Fanuc TP program (LS listing): hs_ov_schraeg2.ls

/PROG  hs_ov_schraeg2
/ATTR
COMMENT	= "18-08-13 11:43:22";
PROG_SIZE	= 0;
DEFAULT_GROUP	= 1, 1, *, *, *;
/APPL
    ARC Welding Equipment: 1, *, *, *, *;
/MN
   1:  CALL HOME_ALL;
   1:  UFRAME_NUM = 1;
   1:  UTOOL_NUM = 3;
   1:  COL GUARD ADJUST 150;
   1:  PR[91] = PR[90];
   1:  ! Sicherheitspunkt;
   1:  PR[92] = PR[90];
   1:  PR[92] = PR[GP1:92,3] + 50;
   1:J PR[92];
   1:  PR[GP1:91,1] = PR[GP1:90,1] + 5.219;
   1:  PR[GP1:91,2] = PR[GP1:90,2] + -0.246;
   1:  PR[GP1:91,3] = PR[GP1:90,3] + 0.915;
   1:L PR[91] 10mm/sec CNT100;
   1:  PR[GP1:91,1] = PR[GP1:90,1] + 8.951;
   1:  PR[GP1:91,2] = PR[GP1:90,2] + -14.614;
   1:L PR[91] 10mm/sec CNT100;
   1:  PR[GP1:91,1] = PR[GP1:90,1] + 8.999;
   1:  PR[GP1:91,2] = PR[GP1:90,2] + -14.812;
   1:L PR[91] 10mm/sec CNT100;
   1:  PR[GP1:91,1] = PR[GP1:90,1] + 9.060;
   1:  PR[GP1:91,2] = PR[GP1:90,2] + -15.209;
   1:L PR[91] 10mm/sec CNT100;
   1:  PR[GP1:91,1] = PR[GP1:90,1] + 9.161;
   1:  PR[GP1:91,2] = PR[GP1:90,2] + -15.468;
   1:L PR[91] 10mm/sec CNT100;
   1:  PR[GP1:91,1] = PR[GP1:90,1] + 18.462;
   1:  PR[GP1:91,2] = PR[GP1:90,2] + -26.550;
   1:L PR[91] 10mm/sec CNT100;
   1:  PR[GP1:91,1] = PR[GP1:90,1] + 18.690;
   1:  PR[GP1:91,2] = PR[GP1:90,2] + -26.887;
   1:L PR[91] 10mm/sec CNT100;
   1:  PR[GP1:91,1] = PR[GP1:90,1] + 18.892;
   1:  PR[GP1:91,2] = PR[GP1:90,2] + -27.077;
   1:L PR[91] 10mm/sec CNT100;
   1:  PR[GP1:91,1] = PR[GP1:90,1] + 32.055;
   1:  PR[GP1:91,2] = PR[GP1:90,2] + -33.088;
   1:L PR[91] 10mm/sec CNT100;
   1:  PR[GP1:91,1] = PR[GP1:90,1] + 32.405;
   1:  PR[GP1:91,2] = PR[GP1:90,2] + -33.295;
   1:L PR[91] 10mm/sec CNT100;
   1:  PR[GP1:91,1] = PR[GP1:90,1] + 32.669;
   1:  PR[GP1:91,2] = PR[GP1:90,2] + -33.380;
   1:L PR[91] 10mm/sec CNT100;
   1:  PR[GP1:91,1] = PR[GP1:90,1] + 47.143;
   1:  PR[GP1:91,2] = PR[GP1:90,2] + -33.149;
   1:L PR[91] 10mm/sec CNT100;
   1:  PR[GP1:91,1] = PR[GP1:90,1] + 47.549;
   1:  PR[GP1:91,2] = PR[GP1:90,2] + -33.186;
   1:L PR[91] 10mm/sec CNT100;
   1:  PR[GP1:91,1] = PR[GP1:90,1] + 47.822;
   1:  PR[GP1:91,2] = PR[GP1:90,2] + -33.150;
   1:L PR[91] 10mm/sec CNT100;
   1:  PR[GP1:91,1] = PR[GP1:90,1] + 60.787;
   1:  PR[GP1:91,2] = PR[GP1:90,2] + -26.722;
   1:L PR[91] 10mm/sec CNT100;
   1:  PR[GP1:91,1] = PR[GP1:90,1] + 61.170;
   1:  PR[GP1:91,2] = PR[GP1:90,2] + -26.581;
   1:L PR[91] 10mm/sec CNT100;
   1:  PR[GP1:91,1] = PR[GP1:90,1] + 61.401;
   1:  PR[GP1:91,2] = PR[GP1:90,2] + -26.432;
   1:L PR[91] 10mm/sec CNT100;
   1:  PR[GP1:91,1] = PR[GP1:90,1] + 70.346;
   1:  PR[GP1:91,2] = PR[GP1:90,2] + -15.058;
   1:L PR[91] 10mm/sec CNT100;
   1:  PR[GP1:91,1] = PR[GP1:90,1] + 70.631;
   1:  PR[GP1:91,2] = PR[GP1:90,2] + -14.767;
   1:L PR[91] 10mm/sec CNT100;
   1:  PR[GP1:91,1] = PR[GP1:90,1] + 70.776;
   1:  PR[GP1:91,2] = PR[GP1:90,2] + -14.533;
   1:L PR[91] 10mm/sec CNT100;
   1:  PR[GP1:91,1] = PR[GP1:90,1] + 73.966;
   1:  PR[GP1:91,2] = PR[GP1:90,2] + -0.414;
   1:L PR[91] 10mm/sec CNT100;
   1:  PR[GP1:91,1] = PR[GP1:90,1] + 74.099;
   1:  PR[GP1:91,2] = PR[GP1:90,2] + -0.028;
   1:L PR[91] 10mm/sec CNT100;
   1:  PR[GP1:91,1] = PR[GP1:90,1] + 74.129;
   1:  PR[GP1:91,2] = PR[GP1:90,2] + 0.245;
   1:L PR[91] 10mm/sec CNT100;
   1:  PR[GP1:91,1] = PR[GP1:90,1] + 70.940;
   1:  PR[GP1:91,2] = PR[GP1:90,2] + 14.363;
   1:L PR[91] 10mm/sec CNT100;
   1:  PR[GP1:91,1] = PR[GP1:90,1] + 70.895;
   1:  PR[GP1:91,2] = PR[GP1:90,2] + 14.770;
   1:L PR[91] 10mm/sec CNT100;
   1:  PR[GP1:91,1] = PR[GP1:90,1] + 70.794;
   1:  PR[GP1:91,2] = PR[GP1:90,2] + 15.062;
   1:L PR[91] 10mm/sec CNT100;
   1:  PR[GP1:91,1] = PR[GP1:90,1] + 70.614;
   1:  PR[GP1:91,2] = PR[GP1:90,2] + 15.353;
   1:L PR[91] 10mm/sec CNT100;
   1:  PR[GP1:91,1] = PR[GP1:90,1] + 61.669;
   1:  PR[GP1:91,2] = PR[GP1:90,2] + 26.727;
   1:L PR[91] 10mm/sec CNT100;
   1:  PR[GP1:91,1] = PR[GP1:90,1] + 61.429;
   1:  PR[GP1:91,2] = PR[GP1:90,2] + 26.972;
   1:L PR[91] 10mm/sec CNT100;
   1:  PR[GP1:91,1] = PR[GP1:90,1] + 61.143;
   1:  PR[GP1:91,2] = PR[GP1:90,2] + 27.157;
   1:L PR[91] 10mm/sec CNT100;
   1:  PR[GP1:91,1] = PR[GP1:90,1] + 48.177;
   1:  PR[GP1:91,2] = PR[GP1:90,2] + 33.585;
   1:L PR[91] 10mm/sec CNT100;
   1:  PR[GP1:91,1] = PR[GP1:90,1] + 47.855;
   1:  PR[GP1:91,2] = PR[GP1:90,2] + 33.703;
   1:L PR[91] 10mm/sec CNT100;
   1:  PR[GP1:91,1] = PR[GP1:90,1] + 47.517;
   1:  PR[GP1:91,2] = PR[GP1:90,2] + 33.748;
   1:L PR[91] 10mm/sec CNT100;
   1:  PR[GP1:91,1] = PR[GP1:90,1] + 33.042;
   1:  PR[GP1:91,2] = PR[GP1:90,2] + 33.978;
   1:L PR[91] 10mm/sec CNT100;
   1:  PR[GP1:91,1] = PR[GP1:90,1] + 32.700;
   1:  PR[GP1:91,2] = PR[GP1:90,2] + 33.948;
   1:L PR[91] 10mm/sec CNT100;
   1:  PR[GP1:91,1] = PR[GP1:90,1] + 32.375;
   1:  PR[GP1:91,2] = PR[GP1:90,2] + 33.843;
   1:L PR[91] 10mm/sec CNT100;
   1:  PR[GP1:91,1] = PR[GP1:90,1] + 19.212;
   1:  PR[GP1:91,2] = PR[GP1:90,2] + 27.832;
   1:L PR[91] 10mm/sec CNT100;
   1:  PR[GP1:91,1] = PR[GP1:90,1] + 18.915;
   1:  PR[GP1:91,2] = PR[GP1:90,2] + 27.657;
   1:L PR[91] 10mm/sec CNT100;
   1:  PR[GP1:91,1] = PR[GP1:90,1] + 18.668;
   1:  PR[GP1:91,2] = PR[GP1:90,2] + 27.424;
   1:L PR[91] 10mm/sec CNT100;
   1:  PR[GP1:91,1] = PR[GP1:90,1] + 9.365;
   1:  PR[GP1:91,2] = PR[GP1:90,2] + 16.341;
   1:L PR[91] 10mm/sec CNT100;
   1:  PR[GP1:91,1] = PR[GP1:90,1] + 9.172;
   1:  PR[GP1:91,2] = PR[GP1:90,2] + 16.055;
   1:L PR[91] 10mm/sec CNT100;
   1:  PR[GP1:91,1] = PR[GP1:90,1] + 9.048;
   1:  PR[GP1:91,2] = PR[GP1:90,2] + 15.739;
   1:L PR[91] 10mm/sec CNT100;
   1:  PR[GP1:91,1] = PR[GP1:90,1] + 5.411;
   1:  PR[GP1:91,2] = PR[GP1:90,2] + 1.740;
   1:L PR[91] 10mm/sec CNT100;
   1:  PR[GP1:91,1] = PR[GP1:90,1] + 5.272;
   1:  PR[GP1:91,2] = PR[GP1:90,2] + 0.804;
   1:L PR[91] 10mm/sec CNT100;
   1:  PR[GP1:91,1] = PR[GP1:90,1] + -5.745;
   1:L PR[91] 10mm/sec CNT100;
   1:  PR[GP1:91,1] = PR[GP1:90,1] + -9.477;
   1:  PR[GP1:91,2] = PR[GP1:90,2] + 15.172;
   1:L PR[91] 10mm/sec CNT100;
   1:  PR[GP1:91,1] = PR[GP1:90,1] + -9.525;
   1:  PR[GP1:91,2] = PR[GP1:90,2] + 15.371;
   1:L PR[91] 10mm/sec CNT100;
   1:  PR[GP1:91,1] = PR[GP1:90,1] + -9.586;
   1:  PR[GP1:91,2] = PR[GP1:90,2] + 15.768;
   1:L PR[91] 10mm/sec CNT100;
   1:  PR[GP1:91,1] = PR[GP1:90,1] + -9.687;
   1:  PR[GP1:91,2] = PR[GP1:90,2] + 16.026;
   1:L PR[91] 10mm/sec CNT100;
   1:  PR[GP1:91,1] = PR[GP1:90,1] + -18.989;
   1:  PR[GP1:91,2] = PR[GP1:90,2] + 27.108;
   1:L PR[91] 10mm/sec CNT100;
   1:  PR[GP1:91,1] = PR[GP1:90,1] + -19.217;
   1:  PR[GP1:91,2] = PR[GP1:90,2] + 27.445;
   1:L PR[91] 10mm/sec CNT100;
   1:  PR[GP1:91,1] = PR[GP1:90,1] + -19.418;
   1:  PR[GP1:91,2] = PR[GP1:90,2] + 27.635;
   1:L PR[91] 10mm/sec CNT100;
   1:  PR[GP1:91,1] = PR[GP1:90,1] + -32.581;
   1:  PR[GP1:91,2] = PR[GP1:90,2] + 33.646;
   1:L PR[91] 10mm/sec CNT100;
   1:  PR[GP1:91,1] = PR[GP1:90,1] + -32.932;
   1:  PR[GP1:91,2] = PR[GP1:90,2] + 33.853;
   1:L PR[91] 10mm/sec CNT100;
   1:  PR[GP1:91,1] = PR[GP1:90,1] + -33.195;
   1:  PR[GP1:91,2] = PR[GP1:90,2] + 33.938;
   1:L PR[91] 10mm/sec CNT100;
   1:  PR[GP1:91,1] = PR[GP1:90,1] + -47.669;
   1:  PR[GP1:91,2] = PR[GP1:90,2] + 33.707;
   1:L PR[91] 10mm/sec CNT100;
   1:  PR[GP1:91,1] = PR[GP1:90,1] + -48.075;
   1:  PR[GP1:91,2] = PR[GP1:90,2] + 33.744;
   1:L PR[91] 10mm/sec CNT100;
   1:  PR[GP1:91,1] = PR[GP1:90,1] + -48.349;
   1:  PR[GP1:91,2] = PR[GP1:90,2] + 33.708;
   1:L PR[91] 10mm/sec CNT100;
   1:  PR[GP1:91,1] = PR[GP1:90,1] + -61.314;
   1:  PR[GP1:91,2] = PR[GP1:90,2] + 27.280;
   1:L PR[91] 10mm/sec CNT100;
   1:  PR[GP1:91,1] = PR[GP1:90,1] + -61.696;
   1:  PR[GP1:91,2] = PR[GP1:90,2] + 27.140;
   1:L PR[91] 10mm/sec CNT100;
   1:  PR[GP1:91,1] = PR[GP1:90,1] + -61.928;
   1:  PR[GP1:91,2] = PR[GP1:90,2] + 26.990;
   1:L PR[91] 10mm/sec CNT100;
   1:  PR[GP1:91,1] = PR[GP1:90,1] + -70.872;
   1:  PR[GP1:91,2] = PR[GP1:90,2] + 15.617;
   1:L PR[91] 10mm/sec CNT100;
   1:  PR[GP1:91,1] = PR[GP1:90,1] + -71.158;
   1:  PR[GP1:91,2] = PR[GP1:90,2] + 15.325;
   1:L PR[91] 10mm/sec CNT100;
   1:  PR[GP1:91,1] = PR[GP1:90,1] + -71.303;
   1:  PR[GP1:91,2] = PR[GP1:90,2] + 15.091;
   1:L PR[91] 10mm/sec CNT100;
   1:  PR[GP1:91,1] = PR[GP1:90,1] + -74.492;
   1:  PR[GP1:91,2] = PR[GP1:90,2] + 0.972;
   1:L PR[91] 10mm/sec CNT100;
   1:  PR[GP1:91,1] = PR[GP1:90,1] + -74.625;
   1:  PR[GP1:91,2] = PR[GP1:90,2] + 0.586;
   1:L PR[91] 10mm/sec CNT100;
   1:  PR[GP1:91,1] = PR[GP1:90,1] + -74.656;
   1:  PR[GP1:91,2] = PR[GP1:90,2] + 0.313;
   1:L PR[91] 10mm/sec CNT100;
   1:  PR[GP1:91,1] = PR[GP1:90,1] + -71.466;
   1:  PR[GP1:91,2] = PR[GP1:90,2] + -13.805;
   1:L PR[91] 10mm/sec CNT100;
   1:  PR[GP1:91,1] = PR[GP1:90,1] + -71.421;
   1:  PR[GP1:91,2] = PR[GP1:90,2] + -14.212;
   1:L PR[91] 10mm/sec CNT100;
   1:  PR[GP1:91,1] = PR[GP1:90,1] + -71.320;
   1:  PR[GP1:91,2] = PR[GP1:90,2] + -14.504;
   1:L PR[91] 10mm/sec CNT100;
   1:  PR[GP1:91,1] = PR[GP1:90,1] + -71.141;
   1:  PR[GP1:91,2] = PR[GP1:90,2] + -14.795;
   1:L PR[91] 10mm/sec CNT100;
   1:  PR[GP1:91,1] = PR[GP1:90,1] + -62.196;
   1:  PR[GP1:91,2] = PR[GP1:90,2] + -26.169;
   1:L PR[91] 10mm/sec CNT100;
   1:  PR[GP1:91,1] = PR[GP1:90,1] + -61.956;
   1:  PR[GP1:91,2] = PR[GP1:90,2] + -26.414;
   1:L PR[91] 10mm/sec CNT100;
   1:  PR[GP1:91,1] = PR[GP1:90,1] + -61.669;
   1:  PR[GP1:91,2] = PR[GP1:90,2] + -26.599;
   1:L PR[91] 10mm/sec CNT100;
   1:  PR[GP1:91,1] = PR[GP1:90,1] + -48.703;
   1:  PR[GP1:91,2] = PR[GP1:90,2] + -33.027;
   1:L PR[91] 10mm/sec CNT100;
   1:  PR[GP1:91,1] = PR[GP1:90,1] + -48.381;
   1:  PR[GP1:91,2] = PR[GP1:90,2] + -33.145;
   1:L PR[91] 10mm/sec CNT100;
   1:  PR[GP1:91,1] = PR[GP1:90,1] + -48.043;
   1:  PR[GP1:91,2] = PR[GP1:90,2] + -33.190;
   1:L PR[91] 10mm/sec CNT100;
   1:  PR[GP1:91,1] = PR[GP1:90,1] + -33.568;
   1:  PR[GP1:91,2] = PR[GP1:90,2] + -33.420;
   1:L PR[91] 10mm/sec CNT100;
   1:  PR[GP1:91,1] = PR[GP1:90,1] + -33.226;
   1:  PR[GP1:91,2] = PR[GP1:90,2] + -33.390;
   1:L PR[91] 10mm/sec CNT100;
   1:  PR[GP1:91,1] = PR[GP1:90,1] + -32.902;
   1:  PR[GP1:91,2] = PR[GP1:90,2] + -33.285;
   1:L PR[91] 10mm/sec CNT100;
   1:  PR[GP1:91,1] = PR[GP1:90,1] + -19.738;
   1:  PR[GP1:91,2] = PR[GP1:90,2] + -27.274;
   1:L PR[91] 10mm/sec CNT100;
   1:  PR[GP1:91,1] = PR[GP1:90,1] + -19.442;
   1:  PR[GP1:91,2] = PR[GP1:90,2] + -27.099;
   1:L PR[91] 10mm/sec CNT100;
   1:  PR[GP1:91,1] = PR[GP1:90,1] + -19.194;
   1:  PR[GP1:91,2] = PR[GP1:90,2] + -26.866;
   1:L PR[91] 10mm/sec CNT100;
   1:  PR[GP1:91,1] = PR[GP1:90,1] + -9.892;
   1:  PR[GP1:91,2] = PR[GP1:90,2] + -15.783;
   1:L PR[91] 10mm/sec CNT100;
   1:  PR[GP1:91,1] = PR[GP1:90,1] + -9.699;
   1:  PR[GP1:91,2] = PR[GP1:90,2] + -15.497;
   1:L PR[91] 10mm/sec CNT100;
   1:  PR[GP1:91,1] = PR[GP1:90,1] + -9.575;
   1:  PR[GP1:91,2] = PR[GP1:90,2] + -15.181;
   1:L PR[91] 10mm/sec CNT100;
   1:  PR[GP1:91,1] = PR[GP1:90,1] + -5.938;
   1:  PR[GP1:91,2] = PR[GP1:90,2] + -1.182;
   1:L PR[91] 10mm/sec CNT100;
   1:  PR[GP1:91,1] = PR[GP1:90,1] + -5.799;
   1:  PR[GP1:91,2] = PR[GP1:90,2] + -0.246;
   1:L PR[91] 10mm/sec CNT100;
   1:  PR[GP1:91,1] = PR[GP1:90,1] + 5.219;
   1:L PR[91] 10mm/sec CNT100;
   1:  PR[GP1:91,1] = PR[GP1:90,1] + 8.514;
   1:  PR[GP1:91,2] = PR[GP1:90,2] + -12.941;
   1:  PR[GP1:91,3] = PR[GP1:90,3] + 1.525;
   1:L PR[91] 10mm/sec CNT100;
   1:  PR[GP1:91,1] = PR[GP1:90,1] + 8.631;
   1:  PR[GP1:91,2] = PR[GP1:90,2] + -13.421;
   1:L PR[91] 10mm/sec CNT100;
   1:  PR[GP1:91,1] = PR[GP1:90,1] + 8.803;
   1:  PR[GP1:91,2] = PR[GP1:90,2] + -14.547;
   1:L PR[91] 10mm/sec CNT100;
   1:  PR[GP1:91,1] = PR[GP1:90,1] + 9.173;
   1:  PR[GP1:91,2] = PR[GP1:90,2] + -15.491;
   1:L PR[91] 10mm/sec CNT100;
   1:  PR[GP1:91,1] = PR[GP1:90,1] + 17.530;
   1:  PR[GP1:91,2] = PR[GP1:90,2] + -25.448;
   1:L PR[91] 10mm/sec CNT100;
   1:  PR[GP1:91,1] = PR[GP1:90,1] + 18.171;
   1:  PR[GP1:91,2] = PR[GP1:90,2] + -26.396;
   1:L PR[91] 10mm/sec CNT100;
   1:  PR[GP1:91,1] = PR[GP1:90,1] + 18.910;
   1:  PR[GP1:91,2] = PR[GP1:90,2] + -27.090;
   1:L PR[91] 10mm/sec CNT100;
   1:  PR[GP1:91,1] = PR[GP1:90,1] + 30.736;
   1:  PR[GP1:91,2] = PR[GP1:90,2] + -32.491;
   1:L PR[91] 10mm/sec CNT100;
   1:  PR[GP1:91,1] = PR[GP1:90,1] + 31.721;
   1:  PR[GP1:91,2] = PR[GP1:90,2] + -33.072;
   1:L PR[91] 10mm/sec CNT100;
   1:  PR[GP1:91,1] = PR[GP1:90,1] + 32.686;
   1:  PR[GP1:91,2] = PR[GP1:90,2] + -33.383;
   1:L PR[91] 10mm/sec CNT100;
   1:  PR[GP1:91,1] = PR[GP1:90,1] + 45.690;
   1:  PR[GP1:91,2] = PR[GP1:90,2] + -33.176;
   1:L PR[91] 10mm/sec CNT100;
   1:  PR[GP1:91,1] = PR[GP1:90,1] + 46.831;
   1:  PR[GP1:91,2] = PR[GP1:90,2] + -33.279;
   1:L PR[91] 10mm/sec CNT100;
   1:  PR[GP1:91,1] = PR[GP1:90,1] + 47.835;
   1:  PR[GP1:91,2] = PR[GP1:90,2] + -33.147;
   1:L PR[91] 10mm/sec CNT100;
   1:  PR[GP1:91,1] = PR[GP1:90,1] + 59.483;
   1:  PR[GP1:91,2] = PR[GP1:90,2] + -27.372;
   1:L PR[91] 10mm/sec CNT100;
   1:  PR[GP1:91,1] = PR[GP1:90,1] + 60.558;
   1:  PR[GP1:91,2] = PR[GP1:90,2] + -26.976;
   1:L PR[91] 10mm/sec CNT100;
   1:  PR[GP1:91,1] = PR[GP1:90,1] + 61.408;
   1:  PR[GP1:91,2] = PR[GP1:90,2] + -26.426;
   1:L PR[91] 10mm/sec CNT100;
   1:  PR[GP1:91,1] = PR[GP1:90,1] + 69.444;
   1:  PR[GP1:91,2] = PR[GP1:90,2] + -16.208;
   1:L PR[91] 10mm/sec CNT100;
   1:  PR[GP1:91,1] = PR[GP1:90,1] + 70.246;
   1:  PR[GP1:91,2] = PR[GP1:90,2] + -15.390;
   1:L PR[91] 10mm/sec CNT100;
   1:  PR[GP1:91,1] = PR[GP1:90,1] + 70.778;
   1:  PR[GP1:91,2] = PR[GP1:90,2] + -14.528;
   1:L PR[91] 10mm/sec CNT100;
   1:  PR[GP1:91,1] = PR[GP1:90,1] + 73.644;
   1:  PR[GP1:91,2] = PR[GP1:90,2] + -1.844;
   1:L PR[91] 10mm/sec CNT100;
   1:  PR[GP1:91,1] = PR[GP1:90,1] + 74.018;
   1:  PR[GP1:91,2] = PR[GP1:90,2] + -0.761;
   1:L PR[91] 10mm/sec CNT100;
   1:  PR[GP1:91,1] = PR[GP1:90,1] + 74.129;
   1:  PR[GP1:91,2] = PR[GP1:90,2] + 0.245;
   1:L PR[91] 10mm/sec CNT100;
   1:  PR[GP1:91,1] = PR[GP1:90,1] + 71.264;
   1:  PR[GP1:91,2] = PR[GP1:90,2] + 12.930;
   1:L PR[91] 10mm/sec CNT100;
   1:  PR[GP1:91,1] = PR[GP1:90,1] + 71.137;
   1:  PR[GP1:91,2] = PR[GP1:90,2] + 14.069;
   1:L PR[91] 10mm/sec CNT100;
   1:  PR[GP1:91,1] = PR[GP1:90,1] + 70.796;
   1:  PR[GP1:91,2] = PR[GP1:90,2] + 15.058;
   1:L PR[91] 10mm/sec CNT100;
   1:  PR[GP1:91,1] = PR[GP1:90,1] + 70.229;
   1:  PR[GP1:91,2] = PR[GP1:90,2] + 15.976;
   1:L PR[91] 10mm/sec CNT100;
   1:  PR[GP1:91,1] = PR[GP1:90,1] + 62.192;
   1:  PR[GP1:91,2] = PR[GP1:90,2] + 26.195;
   1:L PR[91] 10mm/sec CNT100;
   1:  PR[GP1:91,1] = PR[GP1:90,1] + 61.436;
   1:  PR[GP1:91,2] = PR[GP1:90,2] + 26.966;
   1:L PR[91] 10mm/sec CNT100;
   1:  PR[GP1:91,1] = PR[GP1:90,1] + 60.531;
   1:  PR[GP1:91,2] = PR[GP1:90,2] + 27.552;
   1:L PR[91] 10mm/sec CNT100;
   1:  PR[GP1:91,1] = PR[GP1:90,1] + 48.882;
   1:  PR[GP1:91,2] = PR[GP1:90,2] + 33.327;
   1:L PR[91] 10mm/sec CNT100;
   1:  PR[GP1:91,1] = PR[GP1:90,1] + 47.868;
   1:  PR[GP1:91,2] = PR[GP1:90,2] + 33.700;
   1:L PR[91] 10mm/sec CNT100;
   1:  PR[GP1:91,1] = PR[GP1:90,1] + 46.799;
   1:  PR[GP1:91,2] = PR[GP1:90,2] + 33.842;
   1:L PR[91] 10mm/sec CNT100;
   1:  PR[GP1:91,1] = PR[GP1:90,1] + 33.794;
   1:  PR[GP1:91,2] = PR[GP1:90,2] + 34.049;
   1:L PR[91] 10mm/sec CNT100;
   1:  PR[GP1:91,1] = PR[GP1:90,1] + 32.717;
   1:  PR[GP1:91,2] = PR[GP1:90,2] + 33.951;
   1:L PR[91] 10mm/sec CNT100;
   1:  PR[GP1:91,1] = PR[GP1:90,1] + 31.691;
   1:  PR[GP1:91,2] = PR[GP1:90,2] + 33.621;
   1:L PR[91] 10mm/sec CNT100;
   1:  PR[GP1:91,1] = PR[GP1:90,1] + 19.865;
   1:  PR[GP1:91,2] = PR[GP1:90,2] + 28.220;
   1:L PR[91] 10mm/sec CNT100;
   1:  PR[GP1:91,1] = PR[GP1:90,1] + 18.933;
   1:  PR[GP1:91,2] = PR[GP1:90,2] + 27.670;
   1:L PR[91] 10mm/sec CNT100;
   1:  PR[GP1:91,1] = PR[GP1:90,1] + 18.148;
   1:  PR[GP1:91,2] = PR[GP1:90,2] + 26.932;
   1:L PR[91] 10mm/sec CNT100;
   1:  PR[GP1:91,1] = PR[GP1:90,1] + 9.791;
   1:  PR[GP1:91,2] = PR[GP1:90,2] + 16.975;
   1:L PR[91] 10mm/sec CNT100;
   1:  PR[GP1:91,1] = PR[GP1:90,1] + 9.185;
   1:  PR[GP1:91,2] = PR[GP1:90,2] + 16.079;
   1:L PR[91] 10mm/sec CNT100;
   1:  PR[GP1:91,1] = PR[GP1:90,1] + 8.792;
   1:  PR[GP1:91,2] = PR[GP1:90,2] + 15.076;
   1:L PR[91] 10mm/sec CNT100;
   1:  PR[GP1:91,1] = PR[GP1:90,1] + 5.524;
   1:  PR[GP1:91,2] = PR[GP1:90,2] + 2.499;
   1:L PR[91] 10mm/sec CNT100;
   1:  PR[GP1:91,1] = PR[GP1:90,1] + 5.272;
   1:  PR[GP1:91,2] = PR[GP1:90,2] + 0.804;
   1:L PR[91] 10mm/sec CNT100;
   1:  PR[GP1:91,1] = PR[GP1:90,1] + -5.745;
   1:L PR[91] 10mm/sec CNT100;
   1:  PR[GP1:91,1] = PR[GP1:90,1] + -9.040;
   1:  PR[GP1:91,2] = PR[GP1:90,2] + 13.499;
   1:L PR[91] 10mm/sec CNT100;
   1:  PR[GP1:91,1] = PR[GP1:90,1] + -9.157;
   1:  PR[GP1:91,2] = PR[GP1:90,2] + 13.979;
   1:L PR[91] 10mm/sec CNT100;
   1:  PR[GP1:91,1] = PR[GP1:90,1] + -9.329;
   1:  PR[GP1:91,2] = PR[GP1:90,2] + 15.105;
   1:L PR[91] 10mm/sec CNT100;
   1:  PR[GP1:91,1] = PR[GP1:90,1] + -9.699;
   1:  PR[GP1:91,2] = PR[GP1:90,2] + 16.049;
   1:L PR[91] 10mm/sec CNT100;
   1:  PR[GP1:91,1] = PR[GP1:90,1] + -18.056;
   1:  PR[GP1:91,2] = PR[GP1:90,2] + 26.006;
   1:L PR[91] 10mm/sec CNT100;
   1:  PR[GP1:91,1] = PR[GP1:90,1] + -18.697;
   1:  PR[GP1:91,2] = PR[GP1:90,2] + 26.954;
   1:L PR[91] 10mm/sec CNT100;
   1:  PR[GP1:91,1] = PR[GP1:90,1] + -19.436;
   1:  PR[GP1:91,2] = PR[GP1:90,2] + 27.648;
   1:L PR[91] 10mm/sec CNT100;
   1:  PR[GP1:91,1] = PR[GP1:90,1] + -31.262;
   1:  PR[GP1:91,2] = PR[GP1:90,2] + 33.049;
   1:L PR[91] 10mm/sec CNT100;
   1:  PR[GP1:91,1] = PR[GP1:90,1] + -32.248;
   1:  PR[GP1:91,2] = PR[GP1:90,2] + 33.631;
   1:L PR[91] 10mm/sec CNT100;
   1:  PR[GP1:91,1] = PR[GP1:90,1] + -33.213;
   1:  PR[GP1:91,2] = PR[GP1:90,2] + 33.941;
   1:L PR[91] 10mm/sec CNT100;
   1:  PR[GP1:91,1] = PR[GP1:90,1] + -46.217;
   1:  PR[GP1:91,2] = PR[GP1:90,2] + 33.734;
   1:L PR[91] 10mm/sec CNT100;
   1:  PR[GP1:91,1] = PR[GP1:90,1] + -47.357;
   1:  PR[GP1:91,2] = PR[GP1:90,2] + 33.837;
   1:L PR[91] 10mm/sec CNT100;
   1:  PR[GP1:91,1] = PR[GP1:90,1] + -48.361;
   1:  PR[GP1:91,2] = PR[GP1:90,2] + 33.705;
   1:L PR[91] 10mm/sec CNT100;
   1:  PR[GP1:91,1] = PR[GP1:90,1] + -60.010;
   1:  PR[GP1:91,2] = PR[GP1:90,2] + 27.930;
   1:L PR[91] 10mm/sec CNT100;
   1:  PR[GP1:91,1] = PR[GP1:90,1] + -61.084;
   1:  PR[GP1:91,2] = PR[GP1:90,2] + 27.534;
   1:L PR[91] 10mm/sec CNT100;
   1:  PR[GP1:91,1] = PR[GP1:90,1] + -61.935;
   1:  PR[GP1:91,2] = PR[GP1:90,2] + 26.984;
   1:L PR[91] 10mm/sec CNT100;
   1:  PR[GP1:91,1] = PR[GP1:90,1] + -69.971;
   1:  PR[GP1:91,2] = PR[GP1:90,2] + 16.766;
   1:L PR[91] 10mm/sec CNT100;
   1:  PR[GP1:91,1] = PR[GP1:90,1] + -70.772;
   1:  PR[GP1:91,2] = PR[GP1:90,2] + 15.948;
   1:L PR[91] 10mm/sec CNT100;
   1:  PR[GP1:91,1] = PR[GP1:90,1] + -71.305;
   1:  PR[GP1:91,2] = PR[GP1:90,2] + 15.087;
   1:L PR[91] 10mm/sec CNT100;
   1:  PR[GP1:91,1] = PR[GP1:90,1] + -74.170;
   1:  PR[GP1:91,2] = PR[GP1:90,2] + 2.402;
   1:L PR[91] 10mm/sec CNT100;
   1:  PR[GP1:91,1] = PR[GP1:90,1] + -74.544;
   1:  PR[GP1:91,2] = PR[GP1:90,2] + 1.319;
   1:L PR[91] 10mm/sec CNT100;
   1:  PR[GP1:91,1] = PR[GP1:90,1] + -74.656;
   1:  PR[GP1:91,2] = PR[GP1:90,2] + 0.313;
   1:L PR[91] 10mm/sec CNT100;
   1:  PR[GP1:91,1] = PR[GP1:90,1] + -71.790;
   1:  PR[GP1:91,2] = PR[GP1:90,2] + -12.371;
   1:L PR[91] 10mm/sec CNT100;
   1:  PR[GP1:91,1] = PR[GP1:90,1] + -71.663;
   1:  PR[GP1:91,2] = PR[GP1:90,2] + -13.511;
   1:L PR[91] 10mm/sec CNT100;
   1:  PR[GP1:91,1] = PR[GP1:90,1] + -71.322;
   1:  PR[GP1:91,2] = PR[GP1:90,2] + -14.500;
   1:L PR[91] 10mm/sec CNT100;
   1:  PR[GP1:91,1] = PR[GP1:90,1] + -70.755;
   1:  PR[GP1:91,2] = PR[GP1:90,2] + -15.418;
   1:L PR[91] 10mm/sec CNT100;
   1:  PR[GP1:91,1] = PR[GP1:90,1] + -62.719;
   1:  PR[GP1:91,2] = PR[GP1:90,2] + -25.636;
   1:L PR[91] 10mm/sec CNT100;
   1:  PR[GP1:91,1] = PR[GP1:90,1] + -61.963;
   1:  PR[GP1:91,2] = PR[GP1:90,2] + -26.408;
   1:L PR[91] 10mm/sec CNT100;
   1:  PR[GP1:91,1] = PR[GP1:90,1] + -61.057;
   1:  PR[GP1:91,2] = PR[GP1:90,2] + -26.994;
   1:L PR[91] 10mm/sec CNT100;
   1:  PR[GP1:91,1] = PR[GP1:90,1] + -49.408;
   1:  PR[GP1:91,2] = PR[GP1:90,2] + -32.769;
   1:L PR[91] 10mm/sec CNT100;
   1:  PR[GP1:91,1] = PR[GP1:90,1] + -48.394;
   1:  PR[GP1:91,2] = PR[GP1:90,2] + -33.142;
   1:L PR[91] 10mm/sec CNT100;
   1:  PR[GP1:91,1] = PR[GP1:90,1] + -47.325;
   1:  PR[GP1:91,2] = PR[GP1:90,2] + -33.283;
   1:L PR[91] 10mm/sec CNT100;
   1:  PR[GP1:91,1] = PR[GP1:90,1] + -34.320;
   1:  PR[GP1:91,2] = PR[GP1:90,2] + -33.490;
   1:L PR[91] 10mm/sec CNT100;
   1:  PR[GP1:91,1] = PR[GP1:90,1] + -33.244;
   1:  PR[GP1:91,2] = PR[GP1:90,2] + -33.393;
   1:L PR[91] 10mm/sec CNT100;
   1:  PR[GP1:91,1] = PR[GP1:90,1] + -32.218;
   1:  PR[GP1:91,2] = PR[GP1:90,2] + -33.063;
   1:L PR[91] 10mm/sec CNT100;
   1:  PR[GP1:91,1] = PR[GP1:90,1] + -20.391;
   1:  PR[GP1:91,2] = PR[GP1:90,2] + -27.662;
   1:L PR[91] 10mm/sec CNT100;
   1:  PR[GP1:91,1] = PR[GP1:90,1] + -19.460;
   1:  PR[GP1:91,2] = PR[GP1:90,2] + -27.112;
   1:L PR[91] 10mm/sec CNT100;
   1:  PR[GP1:91,1] = PR[GP1:90,1] + -18.675;
   1:  PR[GP1:91,2] = PR[GP1:90,2] + -26.374;
   1:L PR[91] 10mm/sec CNT100;
   1:  PR[GP1:91,1] = PR[GP1:90,1] + -10.317;
   1:  PR[GP1:91,2] = PR[GP1:90,2] + -16.417;
   1:L PR[91] 10mm/sec CNT100;
   1:  PR[GP1:91,1] = PR[GP1:90,1] + -9.711;
   1:  PR[GP1:91,2] = PR[GP1:90,2] + -15.521;
   1:L PR[91] 10mm/sec CNT100;
   1:  PR[GP1:91,1] = PR[GP1:90,1] + -9.318;
   1:  PR[GP1:91,2] = PR[GP1:90,2] + -14.518;
   1:L PR[91] 10mm/sec CNT100;
   1:  PR[GP1:91,1] = PR[GP1:90,1] + -6.050;
   1:  PR[GP1:91,2] = PR[GP1:90,2] + -1.940;
   1:L PR[91] 10mm/sec CNT100;
   1:  PR[GP1:91,1] = PR[GP1:90,1] + -5.799;
   1:  PR[GP1:91,2] = PR[GP1:90,2] + -0.246;
   1:L PR[91] 10mm/sec CNT100;
   1:  PR[GP1:91,1] = PR[GP1:90,1] + 5.219;
   1:L PR[91] 10mm/sec CNT100;
   1:  PR[GP1:91,1] = PR[GP1:90,1] + 8.164;
   1:  PR[GP1:91,2] = PR[GP1:90,2] + -11.602;
   1:  PR[GP1:91,3] = PR[GP1:90,3] + 2.135;
   1:L PR[91] 10mm/sec CNT100;
   1:  PR[GP1:91,1] = PR[GP1:90,1] + 8.336;
   1:  PR[GP1:91,2] = PR[GP1:90,2] + -12.307;
   1:L PR[91] 10mm/sec CNT100;
   1:  PR[GP1:91,1] = PR[GP1:90,1] + 8.598;
   1:  PR[GP1:91,2] = PR[GP1:90,2] + -14.016;
   1:L PR[91] 10mm/sec CNT100;
   1:  PR[GP1:91,1] = PR[GP1:90,1] + 9.183;
   1:  PR[GP1:91,2] = PR[GP1:90,2] + -15.510;
   1:L PR[91] 10mm/sec CNT100;
   1:  PR[GP1:91,1] = PR[GP1:90,1] + 16.784;
   1:  PR[GP1:91,2] = PR[GP1:90,2] + -24.567;
   1:L PR[91] 10mm/sec CNT100;
   1:  PR[GP1:91,1] = PR[GP1:90,1] + 17.756;
   1:  PR[GP1:91,2] = PR[GP1:90,2] + -26.002;
   1:L PR[91] 10mm/sec CNT100;
   1:  PR[GP1:91,1] = PR[GP1:90,1] + 18.924;
   1:  PR[GP1:91,2] = PR[GP1:90,2] + -27.101;
   1:L PR[91] 10mm/sec CNT100;
   1:  PR[GP1:91,1] = PR[GP1:90,1] + 29.681;
   1:  PR[GP1:91,2] = PR[GP1:90,2] + -32.013;
   1:L PR[91] 10mm/sec CNT100;
   1:  PR[GP1:91,1] = PR[GP1:90,1] + 31.174;
   1:  PR[GP1:91,2] = PR[GP1:90,2] + -32.895;
   1:L PR[91] 10mm/sec CNT100;
   1:  PR[GP1:91,1] = PR[GP1:90,1] + 32.701;
   1:  PR[GP1:91,2] = PR[GP1:90,2] + -33.386;
   1:L PR[91] 10mm/sec CNT100;
   1:  PR[GP1:91,1] = PR[GP1:90,1] + 44.529;
   1:  PR[GP1:91,2] = PR[GP1:90,2] + -33.198;
   1:L PR[91] 10mm/sec CNT100;
   1:  PR[GP1:91,1] = PR[GP1:90,1] + 46.256;
   1:  PR[GP1:91,2] = PR[GP1:90,2] + -33.354;
   1:L PR[91] 10mm/sec CNT100;
   1:  PR[GP1:91,1] = PR[GP1:90,1] + 47.845;
   1:  PR[GP1:91,2] = PR[GP1:90,2] + -33.144;
   1:L PR[91] 10mm/sec CNT100;
   1:  PR[GP1:91,1] = PR[GP1:90,1] + 58.440;
   1:  PR[GP1:91,2] = PR[GP1:90,2] + -27.892;
   1:L PR[91] 10mm/sec CNT100;
   1:  PR[GP1:91,1] = PR[GP1:90,1] + 60.068;
   1:  PR[GP1:91,2] = PR[GP1:90,2] + -27.292;
   1:L PR[91] 10mm/sec CNT100;
   1:  PR[GP1:91,1] = PR[GP1:90,1] + 61.414;
   1:  PR[GP1:91,2] = PR[GP1:90,2] + -26.422;
   1:L PR[91] 10mm/sec CNT100;
   1:  PR[GP1:91,1] = PR[GP1:90,1] + 68.723;
   1:  PR[GP1:91,2] = PR[GP1:90,2] + -17.128;
   1:L PR[91] 10mm/sec CNT100;
   1:  PR[GP1:91,1] = PR[GP1:90,1] + 69.937;
   1:  PR[GP1:91,2] = PR[GP1:90,2] + -15.888;
   1:L PR[91] 10mm/sec CNT100;
   1:  PR[GP1:91,1] = PR[GP1:90,1] + 70.780;
   1:  PR[GP1:91,2] = PR[GP1:90,2] + -14.525;
   1:L PR[91] 10mm/sec CNT100;
   1:  PR[GP1:91,1] = PR[GP1:90,1] + 73.386;
   1:  PR[GP1:91,2] = PR[GP1:90,2] + -2.988;
   1:L PR[91] 10mm/sec CNT100;
   1:  PR[GP1:91,1] = PR[GP1:90,1] + 73.952;
   1:  PR[GP1:91,2] = PR[GP1:90,2] + -1.347;
   1:L PR[91] 10mm/sec CNT100;
   1:  PR[GP1:91,1] = PR[GP1:90,1] + 74.129;
   1:  PR[GP1:91,2] = PR[GP1:90,2] + 0.245;
   1:L PR[91] 10mm/sec CNT100;
   1:  PR[GP1:91,1] = PR[GP1:90,1] + 71.523;
   1:  PR[GP1:91,2] = PR[GP1:90,2] + 11.782;
   1:L PR[91] 10mm/sec CNT100;
   1:  PR[GP1:91,1] = PR[GP1:90,1] + 71.331;
   1:  PR[GP1:91,2] = PR[GP1:90,2] + 13.508;
   1:L PR[91] 10mm/sec CNT100;
   1:  PR[GP1:91,1] = PR[GP1:90,1] + 70.798;
   1:  PR[GP1:91,2] = PR[GP1:90,2] + 15.055;
   1:L PR[91] 10mm/sec CNT100;
   1:  PR[GP1:91,1] = PR[GP1:90,1] + 69.920;
   1:  PR[GP1:91,2] = PR[GP1:90,2] + 16.474;
   1:L PR[91] 10mm/sec CNT100;
   1:  PR[GP1:91,1] = PR[GP1:90,1] + 62.610;
   1:  PR[GP1:91,2] = PR[GP1:90,2] + 25.769;
   1:L PR[91] 10mm/sec CNT100;
   1:  PR[GP1:91,1] = PR[GP1:90,1] + 61.442;
   1:  PR[GP1:91,2] = PR[GP1:90,2] + 26.962;
   1:L PR[91] 10mm/sec CNT100;
   1:  PR[GP1:91,1] = PR[GP1:90,1] + 60.041;
   1:  PR[GP1:91,2] = PR[GP1:90,2] + 27.868;
   1:L PR[91] 10mm/sec CNT100;
   1:  PR[GP1:91,1] = PR[GP1:90,1] + 49.446;
   1:  PR[GP1:91,2] = PR[GP1:90,2] + 33.121;
   1:L PR[91] 10mm/sec CNT100;
   1:  PR[GP1:91,1] = PR[GP1:90,1] + 47.878;
   1:  PR[GP1:91,2] = PR[GP1:90,2] + 33.698;
   1:L PR[91] 10mm/sec CNT100;
   1:  PR[GP1:91,1] = PR[GP1:90,1] + 46.224;
   1:  PR[GP1:91,2] = PR[GP1:90,2] + 33.916;
   1:L PR[91] 10mm/sec CNT100;
   1:  PR[GP1:91,1] = PR[GP1:90,1] + 34.395;
   1:  PR[GP1:91,2] = PR[GP1:90,2] + 34.105;
   1:L PR[91] 10mm/sec CNT100;
   1:  PR[GP1:91,1] = PR[GP1:90,1] + 32.731;
   1:  PR[GP1:91,2] = PR[GP1:90,2] + 33.954;
   1:L PR[91] 10mm/sec CNT100;
   1:  PR[GP1:91,1] = PR[GP1:90,1] + 31.144;
   1:  PR[GP1:91,2] = PR[GP1:90,2] + 33.443;
   1:L PR[91] 10mm/sec CNT100;
   1:  PR[GP1:91,1] = PR[GP1:90,1] + 20.387;
   1:  PR[GP1:91,2] = PR[GP1:90,2] + 28.530;
   1:L PR[91] 10mm/sec CNT100;
   1:  PR[GP1:91,1] = PR[GP1:90,1] + 18.948;
   1:  PR[GP1:91,2] = PR[GP1:90,2] + 27.681;
   1:L PR[91] 10mm/sec CNT100;
   1:  PR[GP1:91,1] = PR[GP1:90,1] + 17.733;
   1:  PR[GP1:91,2] = PR[GP1:90,2] + 26.539;
   1:L PR[91] 10mm/sec CNT100;
   1:  PR[GP1:91,1] = PR[GP1:90,1] + 10.131;
   1:  PR[GP1:91,2] = PR[GP1:90,2] + 17.482;
   1:L PR[91] 10mm/sec CNT100;
   1:  PR[GP1:91,1] = PR[GP1:90,1] + 9.194;
   1:  PR[GP1:91,2] = PR[GP1:90,2] + 16.098;
   1:L PR[91] 10mm/sec CNT100;
   1:  PR[GP1:91,1] = PR[GP1:90,1] + 8.586;
   1:  PR[GP1:91,2] = PR[GP1:90,2] + 14.546;
   1:L PR[91] 10mm/sec CNT100;
   1:  PR[GP1:91,1] = PR[GP1:90,1] + 5.614;
   1:  PR[GP1:91,2] = PR[GP1:90,2] + 3.106;
   1:L PR[91] 10mm/sec CNT100;
   1:  PR[GP1:91,1] = PR[GP1:90,1] + 5.272;
   1:  PR[GP1:91,2] = PR[GP1:90,2] + 0.804;
   1:L PR[91] 10mm/sec CNT100;
   1:  PR[GP1:91,1] = PR[GP1:90,1] + -5.746;
   1:L PR[91] 10mm/sec CNT100;
   1:  PR[GP1:91,1] = PR[GP1:90,1] + -8.691;
   1:  PR[GP1:91,2] = PR[GP1:90,2] + 12.160;
   1:L PR[91] 10mm/sec CNT100;
   1:  PR[GP1:91,1] = PR[GP1:90,1] + -8.862;
   1:  PR[GP1:91,2] = PR[GP1:90,2] + 12.866;
   1:L PR[91] 10mm/sec CNT100;
   1:  PR[GP1:91,1] = PR[GP1:90,1] + -9.124;
   1:  PR[GP1:91,2] = PR[GP1:90,2] + 14.574;
   1:L PR[91] 10mm/sec CNT100;
   1:  PR[GP1:91,1] = PR[GP1:90,1] + -9.709;
   1:  PR[GP1:91,2] = PR[GP1:90,2] + 16.068;
   1:L PR[91] 10mm/sec CNT100;
   1:  PR[GP1:91,1] = PR[GP1:90,1] + -17.310;
   1:  PR[GP1:91,2] = PR[GP1:90,2] + 25.125;
   1:L PR[91] 10mm/sec CNT100;
   1:  PR[GP1:91,1] = PR[GP1:90,1] + -18.282;
   1:  PR[GP1:91,2] = PR[GP1:90,2] + 26.561;
   1:L PR[91] 10mm/sec CNT100;
   1:  PR[GP1:91,1] = PR[GP1:90,1] + -19.451;
   1:  PR[GP1:91,2] = PR[GP1:90,2] + 27.659;
   1:L PR[91] 10mm/sec CNT100;
   1:  PR[GP1:91,1] = PR[GP1:90,1] + -30.207;
   1:  PR[GP1:91,2] = PR[GP1:90,2] + 32.571;
   1:L PR[91] 10mm/sec CNT100;
   1:  PR[GP1:91,1] = PR[GP1:90,1] + -31.701;
   1:  PR[GP1:91,2] = PR[GP1:90,2] + 33.453;
   1:L PR[91] 10mm/sec CNT100;
   1:  PR[GP1:91,1] = PR[GP1:90,1] + -33.227;
   1:  PR[GP1:91,2] = PR[GP1:90,2] + 33.944;
   1:L PR[91] 10mm/sec CNT100;
   1:  PR[GP1:91,1] = PR[GP1:90,1] + -45.055;
   1:  PR[GP1:91,2] = PR[GP1:90,2] + 33.756;
   1:L PR[91] 10mm/sec CNT100;
   1:  PR[GP1:91,1] = PR[GP1:90,1] + -46.782;
   1:  PR[GP1:91,2] = PR[GP1:90,2] + 33.912;
   1:L PR[91] 10mm/sec CNT100;
   1:  PR[GP1:91,1] = PR[GP1:90,1] + -48.372;
   1:  PR[GP1:91,2] = PR[GP1:90,2] + 33.702;
   1:L PR[91] 10mm/sec CNT100;
   1:  PR[GP1:91,1] = PR[GP1:90,1] + -58.966;
   1:  PR[GP1:91,2] = PR[GP1:90,2] + 28.450;
   1:L PR[91] 10mm/sec CNT100;
   1:  PR[GP1:91,1] = PR[GP1:90,1] + -60.595;
   1:  PR[GP1:91,2] = PR[GP1:90,2] + 27.850;
   1:L PR[91] 10mm/sec CNT100;
   1:  PR[GP1:91,1] = PR[GP1:90,1] + -61.940;
   1:  PR[GP1:91,2] = PR[GP1:90,2] + 26.980;
   1:L PR[91] 10mm/sec CNT100;
   1:  PR[GP1:91,1] = PR[GP1:90,1] + -69.249;
   1:  PR[GP1:91,2] = PR[GP1:90,2] + 17.686;
   1:L PR[91] 10mm/sec CNT100;
   1:  PR[GP1:91,1] = PR[GP1:90,1] + -70.464;
   1:  PR[GP1:91,2] = PR[GP1:90,2] + 16.446;
   1:L PR[91] 10mm/sec CNT100;
   1:  PR[GP1:91,1] = PR[GP1:90,1] + -71.306;
   1:  PR[GP1:91,2] = PR[GP1:90,2] + 15.083;
   1:L PR[91] 10mm/sec CNT100;
   1:  PR[GP1:91,1] = PR[GP1:90,1] + -73.913;
   1:  PR[GP1:91,2] = PR[GP1:90,2] + 3.546;
   1:L PR[91] 10mm/sec CNT100;
   1:  PR[GP1:91,1] = PR[GP1:90,1] + -74.479;
   1:  PR[GP1:91,2] = PR[GP1:90,2] + 1.905;
   1:L PR[91] 10mm/sec CNT100;
   1:  PR[GP1:91,1] = PR[GP1:90,1] + -74.656;
   1:  PR[GP1:91,2] = PR[GP1:90,2] + 0.313;
   1:L PR[91] 10mm/sec CNT100;
   1:  PR[GP1:91,1] = PR[GP1:90,1] + -72.049;
   1:  PR[GP1:91,2] = PR[GP1:90,2] + -11.224;
   1:L PR[91] 10mm/sec CNT100;
   1:  PR[GP1:91,1] = PR[GP1:90,1] + -71.857;
   1:  PR[GP1:91,2] = PR[GP1:90,2] + -12.950;
   1:L PR[91] 10mm/sec CNT100;
   1:  PR[GP1:91,1] = PR[GP1:90,1] + -71.324;
   1:  PR[GP1:91,2] = PR[GP1:90,2] + -14.496;
   1:L PR[91] 10mm/sec CNT100;
   1:  PR[GP1:91,1] = PR[GP1:90,1] + -70.446;
   1:  PR[GP1:91,2] = PR[GP1:90,2] + -15.916;
   1:L PR[91] 10mm/sec CNT100;
   1:  PR[GP1:91,1] = PR[GP1:90,1] + -63.137;
   1:  PR[GP1:91,2] = PR[GP1:90,2] + -25.211;
   1:L PR[91] 10mm/sec CNT100;
   1:  PR[GP1:91,1] = PR[GP1:90,1] + -61.968;
   1:  PR[GP1:91,2] = PR[GP1:90,2] + -26.404;
   1:L PR[91] 10mm/sec CNT100;
   1:  PR[GP1:91,1] = PR[GP1:90,1] + -60.567;
   1:  PR[GP1:91,2] = PR[GP1:90,2] + -27.310;
   1:L PR[91] 10mm/sec CNT100;
   1:  PR[GP1:91,1] = PR[GP1:90,1] + -49.972;
   1:  PR[GP1:91,2] = PR[GP1:90,2] + -32.563;
   1:L PR[91] 10mm/sec CNT100;
   1:  PR[GP1:91,1] = PR[GP1:90,1] + -48.404;
   1:  PR[GP1:91,2] = PR[GP1:90,2] + -33.140;
   1:L PR[91] 10mm/sec CNT100;
   1:  PR[GP1:91,1] = PR[GP1:90,1] + -46.751;
   1:  PR[GP1:91,2] = PR[GP1:90,2] + -33.358;
   1:L PR[91] 10mm/sec CNT100;
   1:  PR[GP1:91,1] = PR[GP1:90,1] + -34.922;
   1:  PR[GP1:91,2] = PR[GP1:90,2] + -33.546;
   1:L PR[91] 10mm/sec CNT100;
   1:  PR[GP1:91,1] = PR[GP1:90,1] + -33.258;
   1:  PR[GP1:91,2] = PR[GP1:90,2] + -33.396;
   1:L PR[91] 10mm/sec CNT100;
   1:  PR[GP1:91,1] = PR[GP1:90,1] + -31.670;
   1:  PR[GP1:91,2] = PR[GP1:90,2] + -32.885;
   1:L PR[91] 10mm/sec CNT100;
   1:  PR[GP1:91,1] = PR[GP1:90,1] + -20.913;
   1:  PR[GP1:91,2] = PR[GP1:90,2] + -27.972;
   1:L PR[91] 10mm/sec CNT100;
   1:  PR[GP1:91,1] = PR[GP1:90,1] + -19.474;
   1:  PR[GP1:91,2] = PR[GP1:90,2] + -27.123;
   1:L PR[91] 10mm/sec CNT100;
   1:  PR[GP1:91,1] = PR[GP1:90,1] + -18.259;
   1:  PR[GP1:91,2] = PR[GP1:90,2] + -25.981;
   1:L PR[91] 10mm/sec CNT100;
   1:  PR[GP1:91,1] = PR[GP1:90,1] + -10.657;
   1:  PR[GP1:91,2] = PR[GP1:90,2] + -16.924;
   1:L PR[91] 10mm/sec CNT100;
   1:  PR[GP1:91,1] = PR[GP1:90,1] + -9.721;
   1:  PR[GP1:91,2] = PR[GP1:90,2] + -15.540;
   1:L PR[91] 10mm/sec CNT100;
   1:  PR[GP1:91,1] = PR[GP1:90,1] + -9.113;
   1:  PR[GP1:91,2] = PR[GP1:90,2] + -13.987;
   1:L PR[91] 10mm/sec CNT100;
   1:  PR[GP1:91,1] = PR[GP1:90,1] + -6.141;
   1:  PR[GP1:91,2] = PR[GP1:90,2] + -2.548;
   1:L PR[91] 10mm/sec CNT100;
   1:  PR[GP1:91,1] = PR[GP1:90,1] + -5.799;
   1:  PR[GP1:91,2] = PR[GP1:90,2] + -0.246;
   1:L PR[91] 10mm/sec CNT100;
   1:  PR[GP1:91,1] = PR[GP1:90,1] + 5.219;
   1:L PR[91] 10mm/sec CNT100;
   1:  PR[GP1:91,1] = PR[GP1:90,1] + 7.493;
   1:  PR[GP1:91,2] = PR[GP1:90,2] + -9.001;
   1:  PR[GP1:91,3] = PR[GP1:90,3] + 2.745;
   1:L PR[91] 10mm/sec CNT100;
   1:  PR[GP1:91,1] = PR[GP1:90,1] + 8.041;
   1:  PR[GP1:91,2] = PR[GP1:90,2] + -11.192;
   1:L PR[91] 10mm/sec CNT100;
   1:  PR[GP1:91,1] = PR[GP1:90,1] + 8.392;
   1:  PR[GP1:91,2] = PR[GP1:90,2] + -13.486;
   1:L PR[91] 10mm/sec CNT100;
   1:  PR[GP1:91,1] = PR[GP1:90,1] + 9.193;
   1:  PR[GP1:91,2] = PR[GP1:90,2] + -15.529;
   1:L PR[91] 10mm/sec CNT100;
   1:  PR[GP1:91,1] = PR[GP1:90,1] + 16.038;
   1:  PR[GP1:91,2] = PR[GP1:90,2] + -23.685;
   1:L PR[91] 10mm/sec CNT100;
   1:  PR[GP1:91,1] = PR[GP1:90,1] + 17.340;
   1:  PR[GP1:91,2] = PR[GP1:90,2] + -25.609;
   1:L PR[91] 10mm/sec CNT100;
   1:  PR[GP1:91,1] = PR[GP1:90,1] + 18.938;
   1:  PR[GP1:91,2] = PR[GP1:90,2] + -27.112;
   1:L PR[91] 10mm/sec CNT100;
   1:  PR[GP1:91,1] = PR[GP1:90,1] + 28.625;
   1:  PR[GP1:91,2] = PR[GP1:90,2] + -31.536;
   1:L PR[91] 10mm/sec CNT100;
   1:  PR[GP1:91,1] = PR[GP1:90,1] + 30.627;
   1:  PR[GP1:91,2] = PR[GP1:90,2] + -32.717;
   1:L PR[91] 10mm/sec CNT100;
   1:  PR[GP1:91,1] = PR[GP1:90,1] + 32.715;
   1:  PR[GP1:91,2] = PR[GP1:90,2] + -33.389;
   1:L PR[91] 10mm/sec CNT100;
   1:  PR[GP1:91,1] = PR[GP1:90,1] + 43.367;
   1:  PR[GP1:91,2] = PR[GP1:90,2] + -33.220;
   1:L PR[91] 10mm/sec CNT100;
   1:  PR[GP1:91,1] = PR[GP1:90,1] + 45.682;
   1:  PR[GP1:91,2] = PR[GP1:90,2] + -33.429;
   1:L PR[91] 10mm/sec CNT100;
   1:  PR[GP1:91,1] = PR[GP1:90,1] + 47.856;
   1:  PR[GP1:91,2] = PR[GP1:90,2] + -33.142;
   1:L PR[91] 10mm/sec CNT100;
   1:  PR[GP1:91,1] = PR[GP1:90,1] + 57.397;
   1:  PR[GP1:91,2] = PR[GP1:90,2] + -28.412;
   1:L PR[91] 10mm/sec CNT100;
   1:  PR[GP1:91,1] = PR[GP1:90,1] + 59.579;
   1:  PR[GP1:91,2] = PR[GP1:90,2] + -27.608;
   1:L PR[91] 10mm/sec CNT100;
   1:  PR[GP1:91,1] = PR[GP1:90,1] + 61.419;
   1:  PR[GP1:91,2] = PR[GP1:90,2] + -26.417;
   1:L PR[91] 10mm/sec CNT100;
   1:  PR[GP1:91,1] = PR[GP1:90,1] + 68.002;
   1:  PR[GP1:91,2] = PR[GP1:90,2] + -18.047;
   1:L PR[91] 10mm/sec CNT100;
   1:  PR[GP1:91,1] = PR[GP1:90,1] + 69.629;
   1:  PR[GP1:91,2] = PR[GP1:90,2] + -16.386;
   1:L PR[91] 10mm/sec CNT100;
   1:  PR[GP1:91,1] = PR[GP1:90,1] + 70.781;
   1:  PR[GP1:91,2] = PR[GP1:90,2] + -14.522;
   1:L PR[91] 10mm/sec CNT100;
   1:  PR[GP1:91,1] = PR[GP1:90,1] + 73.129;
   1:  PR[GP1:91,2] = PR[GP1:90,2] + -4.132;
   1:L PR[91] 10mm/sec CNT100;
   1:  PR[GP1:91,1] = PR[GP1:90,1] + 73.887;
   1:  PR[GP1:91,2] = PR[GP1:90,2] + -1.933;
   1:L PR[91] 10mm/sec CNT100;
   1:  PR[GP1:91,1] = PR[GP1:90,1] + 74.129;
   1:  PR[GP1:91,2] = PR[GP1:90,2] + 0.245;
   1:L PR[91] 10mm/sec CNT100;
   1:  PR[GP1:91,1] = PR[GP1:90,1] + 71.782;
   1:  PR[GP1:91,2] = PR[GP1:90,2] + 10.635;
   1:L PR[91] 10mm/sec CNT100;
   1:  PR[GP1:91,1] = PR[GP1:90,1] + 71.525;
   1:  PR[GP1:91,2] = PR[GP1:90,2] + 12.947;
   1:L PR[91] 10mm/sec CNT100;
   1:  PR[GP1:91,1] = PR[GP1:90,1] + 70.799;
   1:  PR[GP1:91,2] = PR[GP1:90,2] + 15.051;
   1:L PR[91] 10mm/sec CNT100;
   1:  PR[GP1:91,1] = PR[GP1:90,1] + 69.612;
   1:  PR[GP1:91,2] = PR[GP1:90,2] + 16.972;
   1:L PR[91] 10mm/sec CNT100;
   1:  PR[GP1:91,1] = PR[GP1:90,1] + 63.029;
   1:  PR[GP1:91,2] = PR[GP1:90,2] + 25.343;
   1:L PR[91] 10mm/sec CNT100;
   1:  PR[GP1:91,1] = PR[GP1:90,1] + 61.447;
   1:  PR[GP1:91,2] = PR[GP1:90,2] + 26.957;
   1:L PR[91] 10mm/sec CNT100;
   1:  PR[GP1:91,1] = PR[GP1:90,1] + 59.551;
   1:  PR[GP1:91,2] = PR[GP1:90,2] + 28.184;
   1:L PR[91] 10mm/sec CNT100;
   1:  PR[GP1:91,1] = PR[GP1:90,1] + 50.009;
   1:  PR[GP1:91,2] = PR[GP1:90,2] + 32.914;
   1:L PR[91] 10mm/sec CNT100;
   1:  PR[GP1:91,1] = PR[GP1:90,1] + 47.888;
   1:  PR[GP1:91,2] = PR[GP1:90,2] + 33.695;
   1:L PR[91] 10mm/sec CNT100;
   1:  PR[GP1:91,1] = PR[GP1:90,1] + 45.650;
   1:  PR[GP1:91,2] = PR[GP1:90,2] + 33.991;
   1:L PR[91] 10mm/sec CNT100;
   1:  PR[GP1:91,1] = PR[GP1:90,1] + 34.997;
   1:  PR[GP1:91,2] = PR[GP1:90,2] + 34.161;
   1:L PR[91] 10mm/sec CNT100;
   1:  PR[GP1:91,1] = PR[GP1:90,1] + 32.746;
   1:  PR[GP1:91,2] = PR[GP1:90,2] + 33.957;
   1:L PR[91] 10mm/sec CNT100;
   1:  PR[GP1:91,1] = PR[GP1:90,1] + 30.597;
   1:  PR[GP1:91,2] = PR[GP1:90,2] + 33.265;
   1:L PR[91] 10mm/sec CNT100;
   1:  PR[GP1:91,1] = PR[GP1:90,1] + 20.909;
   1:  PR[GP1:91,2] = PR[GP1:90,2] + 28.841;
   1:L PR[91] 10mm/sec CNT100;
   1:  PR[GP1:91,1] = PR[GP1:90,1] + 18.962;
   1:  PR[GP1:91,2] = PR[GP1:90,2] + 27.692;
   1:L PR[91] 10mm/sec CNT100;
   1:  PR[GP1:91,1] = PR[GP1:90,1] + 17.317;
   1:  PR[GP1:91,2] = PR[GP1:90,2] + 26.146;
   1:L PR[91] 10mm/sec CNT100;
   1:  PR[GP1:91,1] = PR[GP1:90,1] + 10.471;
   1:  PR[GP1:91,2] = PR[GP1:90,2] + 17.989;
   1:L PR[91] 10mm/sec CNT100;
   1:  PR[GP1:91,1] = PR[GP1:90,1] + 9.204;
   1:  PR[GP1:91,2] = PR[GP1:90,2] + 16.116;
   1:L PR[91] 10mm/sec CNT100;
   1:  PR[GP1:91,1] = PR[GP1:90,1] + 8.381;
   1:  PR[GP1:91,2] = PR[GP1:90,2] + 14.015;
   1:L PR[91] 10mm/sec CNT100;
   1:  PR[GP1:91,1] = PR[GP1:90,1] + 5.704;
   1:  PR[GP1:91,2] = PR[GP1:90,2] + 3.712;
   1:L PR[91] 10mm/sec CNT100;
   1:  PR[GP1:91,1] = PR[GP1:90,1] + 5.357;
   1:  PR[GP1:91,2] = PR[GP1:90,2] + 1.444;
   1:L PR[91] 10mm/sec CNT100;
   1:  PR[GP1:91,1] = PR[GP1:90,1] + 5.333;
   1:  PR[GP1:91,2] = PR[GP1:90,2] + 0.804;
   1:L PR[91] 10mm/sec CNT100;
   1:  PR[GP1:91,1] = PR[GP1:90,1] + -5.745;
   1:L PR[91] 10mm/sec CNT100;
   1:  PR[GP1:91,1] = PR[GP1:90,1] + -8.020;
   1:  PR[GP1:91,2] = PR[GP1:90,2] + 9.559;
   1:L PR[91] 10mm/sec CNT100;
   1:  PR[GP1:91,1] = PR[GP1:90,1] + -8.567;
   1:  PR[GP1:91,2] = PR[GP1:90,2] + 11.750;
   1:L PR[91] 10mm/sec CNT100;
   1:  PR[GP1:91,1] = PR[GP1:90,1] + -8.919;
   1:  PR[GP1:91,2] = PR[GP1:90,2] + 14.044;
   1:L PR[91] 10mm/sec CNT100;
   1:  PR[GP1:91,1] = PR[GP1:90,1] + -9.719;
   1:  PR[GP1:91,2] = PR[GP1:90,2] + 16.087;
   1:L PR[91] 10mm/sec CNT100;
   1:  PR[GP1:91,1] = PR[GP1:90,1] + -16.564;
   1:  PR[GP1:91,2] = PR[GP1:90,2] + 24.243;
   1:L PR[91] 10mm/sec CNT100;
   1:  PR[GP1:91,1] = PR[GP1:90,1] + -17.866;
   1:  PR[GP1:91,2] = PR[GP1:90,2] + 26.167;
   1:L PR[91] 10mm/sec CNT100;
   1:  PR[GP1:91,1] = PR[GP1:90,1] + -19.465;
   1:  PR[GP1:91,2] = PR[GP1:90,2] + 27.670;
   1:L PR[91] 10mm/sec CNT100;
   1:  PR[GP1:91,1] = PR[GP1:90,1] + -29.152;
   1:  PR[GP1:91,2] = PR[GP1:90,2] + 32.094;
   1:L PR[91] 10mm/sec CNT100;
   1:  PR[GP1:91,1] = PR[GP1:90,1] + -31.153;
   1:  PR[GP1:91,2] = PR[GP1:90,2] + 33.275;
   1:L PR[91] 10mm/sec CNT100;
   1:  PR[GP1:91,1] = PR[GP1:90,1] + -33.241;
   1:  PR[GP1:91,2] = PR[GP1:90,2] + 33.947;
   1:L PR[91] 10mm/sec CNT100;
   1:  PR[GP1:91,1] = PR[GP1:90,1] + -43.893;
   1:  PR[GP1:91,2] = PR[GP1:90,2] + 33.778;
   1:L PR[91] 10mm/sec CNT100;
   1:  PR[GP1:91,1] = PR[GP1:90,1] + -46.208;
   1:  PR[GP1:91,2] = PR[GP1:90,2] + 33.987;
   1:L PR[91] 10mm/sec CNT100;
   1:  PR[GP1:91,1] = PR[GP1:90,1] + -48.382;
   1:  PR[GP1:91,2] = PR[GP1:90,2] + 33.700;
   1:L PR[91] 10mm/sec CNT100;
   1:  PR[GP1:91,1] = PR[GP1:90,1] + -57.923;
   1:  PR[GP1:91,2] = PR[GP1:90,2] + 28.970;
   1:L PR[91] 10mm/sec CNT100;
   1:  PR[GP1:91,1] = PR[GP1:90,1] + -60.105;
   1:  PR[GP1:91,2] = PR[GP1:90,2] + 28.166;
   1:L PR[91] 10mm/sec CNT100;
   1:  PR[GP1:91,1] = PR[GP1:90,1] + -61.946;
   1:  PR[GP1:91,2] = PR[GP1:90,2] + 26.975;
   1:L PR[91] 10mm/sec CNT100;
   1:  PR[GP1:91,1] = PR[GP1:90,1] + -68.528;
   1:  PR[GP1:91,2] = PR[GP1:90,2] + 18.605;
   1:L PR[91] 10mm/sec CNT100;
   1:  PR[GP1:91,1] = PR[GP1:90,1] + -70.155;
   1:  PR[GP1:91,2] = PR[GP1:90,2] + 16.944;
   1:L PR[91] 10mm/sec CNT100;
   1:  PR[GP1:91,1] = PR[GP1:90,1] + -71.308;
   1:  PR[GP1:91,2] = PR[GP1:90,2] + 15.080;
   1:L PR[91] 10mm/sec CNT100;
   1:  PR[GP1:91,1] = PR[GP1:90,1] + -73.655;
   1:  PR[GP1:91,2] = PR[GP1:90,2] + 4.690;
   1:L PR[91] 10mm/sec CNT100;
   1:  PR[GP1:91,1] = PR[GP1:90,1] + -74.414;
   1:  PR[GP1:91,2] = PR[GP1:90,2] + 2.491;
   1:L PR[91] 10mm/sec CNT100;
   1:  PR[GP1:91,1] = PR[GP1:90,1] + -74.656;
   1:  PR[GP1:91,2] = PR[GP1:90,2] + 0.313;
   1:L PR[91] 10mm/sec CNT100;
   1:  PR[GP1:91,1] = PR[GP1:90,1] + -72.308;
   1:  PR[GP1:91,2] = PR[GP1:90,2] + -10.077;
   1:L PR[91] 10mm/sec CNT100;
   1:  PR[GP1:91,1] = PR[GP1:90,1] + -72.051;
   1:  PR[GP1:91,2] = PR[GP1:90,2] + -12.389;
   1:L PR[91] 10mm/sec CNT100;
   1:  PR[GP1:91,1] = PR[GP1:90,1] + -71.326;
   1:  PR[GP1:91,2] = PR[GP1:90,2] + -14.493;
   1:L PR[91] 10mm/sec CNT100;
   1:  PR[GP1:91,1] = PR[GP1:90,1] + -70.138;
   1:  PR[GP1:91,2] = PR[GP1:90,2] + -16.414;
   1:L PR[91] 10mm/sec CNT100;
   1:  PR[GP1:91,1] = PR[GP1:90,1] + -63.555;
   1:  PR[GP1:91,2] = PR[GP1:90,2] + -24.785;
   1:L PR[91] 10mm/sec CNT100;
   1:  PR[GP1:91,1] = PR[GP1:90,1] + -61.974;
   1:  PR[GP1:91,2] = PR[GP1:90,2] + -26.399;
   1:L PR[91] 10mm/sec CNT100;
   1:  PR[GP1:91,1] = PR[GP1:90,1] + -60.078;
   1:  PR[GP1:91,2] = PR[GP1:90,2] + -27.626;
   1:L PR[91] 10mm/sec CNT100;
   1:  PR[GP1:91,1] = PR[GP1:90,1] + -50.536;
   1:  PR[GP1:91,2] = PR[GP1:90,2] + -32.356;
   1:L PR[91] 10mm/sec CNT100;
   1:  PR[GP1:91,1] = PR[GP1:90,1] + -48.415;
   1:  PR[GP1:91,2] = PR[GP1:90,2] + -33.137;
   1:L PR[91] 10mm/sec CNT100;
   1:  PR[GP1:91,1] = PR[GP1:90,1] + -46.176;
   1:  PR[GP1:91,2] = PR[GP1:90,2] + -33.433;
   1:L PR[91] 10mm/sec CNT100;
   1:  PR[GP1:91,1] = PR[GP1:90,1] + -35.523;
   1:  PR[GP1:91,2] = PR[GP1:90,2] + -33.602;
   1:L PR[91] 10mm/sec CNT100;
   1:  PR[GP1:91,1] = PR[GP1:90,1] + -33.272;
   1:  PR[GP1:91,2] = PR[GP1:90,2] + -33.399;
   1:L PR[91] 10mm/sec CNT100;
   1:  PR[GP1:91,1] = PR[GP1:90,1] + -31.123;
   1:  PR[GP1:91,2] = PR[GP1:90,2] + -32.707;
   1:L PR[91] 10mm/sec CNT100;
   1:  PR[GP1:91,1] = PR[GP1:90,1] + -21.436;
   1:  PR[GP1:91,2] = PR[GP1:90,2] + -28.283;
   1:L PR[91] 10mm/sec CNT100;
   1:  PR[GP1:91,1] = PR[GP1:90,1] + -19.488;
   1:  PR[GP1:91,2] = PR[GP1:90,2] + -27.134;
   1:L PR[91] 10mm/sec CNT100;
   1:  PR[GP1:91,1] = PR[GP1:90,1] + -17.844;
   1:  PR[GP1:91,2] = PR[GP1:90,2] + -25.588;
   1:L PR[91] 10mm/sec CNT100;
   1:  PR[GP1:91,1] = PR[GP1:90,1] + -10.998;
   1:  PR[GP1:91,2] = PR[GP1:90,2] + -17.431;
   1:L PR[91] 10mm/sec CNT100;
   1:  PR[GP1:91,1] = PR[GP1:90,1] + -9.730;
   1:  PR[GP1:91,2] = PR[GP1:90,2] + -15.558;
   1:L PR[91] 10mm/sec CNT100;
   1:  PR[GP1:91,1] = PR[GP1:90,1] + -8.907;
   1:  PR[GP1:91,2] = PR[GP1:90,2] + -13.457;
   1:L PR[91] 10mm/sec CNT100;
   1:  PR[GP1:91,1] = PR[GP1:90,1] + -6.230;
   1:  PR[GP1:91,2] = PR[GP1:90,2] + -3.154;
   1:L PR[91] 10mm/sec CNT100;
   1:  PR[GP1:91,1] = PR[GP1:90,1] + -5.883;
   1:  PR[GP1:91,2] = PR[GP1:90,2] + -0.886;
   1:L PR[91] 10mm/sec CNT100;
   1:  PR[GP1:91,1] = PR[GP1:90,1] + -5.860;
   1:  PR[GP1:91,2] = PR[GP1:90,2] + -0.246;
   1:L PR[91] 10mm/sec CNT100;
   1:  PR[GP1:91,1] = PR[GP1:90,1] + 5.219;
   1:L PR[91] 10mm/sec CNT100;
   1:  PR[GP1:91,1] = PR[GP1:90,1] + 7.064;
   1:  PR[GP1:91,2] = PR[GP1:90,2] + -7.347;
   1:  PR[GP1:91,3] = PR[GP1:90,3] + 3.355;
   1:L PR[91] 10mm/sec CNT100;
   1:  PR[GP1:91,1] = PR[GP1:90,1] + 7.746;
   1:  PR[GP1:91,2] = PR[GP1:90,2] + -10.079;
   1:L PR[91] 10mm/sec CNT100;
   1:  PR[GP1:91,1] = PR[GP1:90,1] + 8.187;
   1:  PR[GP1:91,2] = PR[GP1:90,2] + -12.956;
   1:L PR[91] 10mm/sec CNT100;
   1:  PR[GP1:91,1] = PR[GP1:90,1] + 9.202;
   1:  PR[GP1:91,2] = PR[GP1:90,2] + -15.548;
   1:L PR[91] 10mm/sec CNT100;
   1:  PR[GP1:91,1] = PR[GP1:90,1] + 15.292;
   1:  PR[GP1:91,2] = PR[GP1:90,2] + -22.803;
   1:L PR[91] 10mm/sec CNT100;
   1:  PR[GP1:91,1] = PR[GP1:90,1] + 16.925;
   1:  PR[GP1:91,2] = PR[GP1:90,2] + -25.216;
   1:L PR[91] 10mm/sec CNT100;
   1:  PR[GP1:91,1] = PR[GP1:90,1] + 18.953;
   1:  PR[GP1:91,2] = PR[GP1:90,2] + -27.123;
   1:L PR[91] 10mm/sec CNT100;
   1:  PR[GP1:91,1] = PR[GP1:90,1] + 27.570;
   1:  PR[GP1:91,2] = PR[GP1:90,2] + -31.058;
   1:L PR[91] 10mm/sec CNT100;
   1:  PR[GP1:91,1] = PR[GP1:90,1] + 30.080;
   1:  PR[GP1:91,2] = PR[GP1:90,2] + -32.539;
   1:L PR[91] 10mm/sec CNT100;
   1:  PR[GP1:91,1] = PR[GP1:90,1] + 32.729;
   1:  PR[GP1:91,2] = PR[GP1:90,2] + -33.392;
   1:L PR[91] 10mm/sec CNT100;
   1:  PR[GP1:91,1] = PR[GP1:90,1] + 42.205;
   1:  PR[GP1:91,2] = PR[GP1:90,2] + -33.241;
   1:L PR[91] 10mm/sec CNT100;
   1:  PR[GP1:91,1] = PR[GP1:90,1] + 45.107;
   1:  PR[GP1:91,2] = PR[GP1:90,2] + -33.503;
   1:L PR[91] 10mm/sec CNT100;
   1:  PR[GP1:91,1] = PR[GP1:90,1] + 47.866;
   1:  PR[GP1:91,2] = PR[GP1:90,2] + -33.139;
   1:L PR[91] 10mm/sec CNT100;
   1:  PR[GP1:91,1] = PR[GP1:90,1] + 56.354;
   1:  PR[GP1:91,2] = PR[GP1:90,2] + -28.931;
   1:L PR[91] 10mm/sec CNT100;
   1:  PR[GP1:91,1] = PR[GP1:90,1] + 59.089;
   1:  PR[GP1:91,2] = PR[GP1:90,2] + -27.924;
   1:L PR[91] 10mm/sec CNT100;
   1:  PR[GP1:91,1] = PR[GP1:90,1] + 61.425;
   1:  PR[GP1:91,2] = PR[GP1:90,2] + -26.413;
   1:L PR[91] 10mm/sec CNT100;
   1:  PR[GP1:91,1] = PR[GP1:90,1] + 67.281;
   1:  PR[GP1:91,2] = PR[GP1:90,2] + -18.967;
   1:L PR[91] 10mm/sec CNT100;
   1:  PR[GP1:91,1] = PR[GP1:90,1] + 69.320;
   1:  PR[GP1:91,2] = PR[GP1:90,2] + -16.885;
   1:L PR[91] 10mm/sec CNT100;
   1:  PR[GP1:91,1] = PR[GP1:90,1] + 70.783;
   1:  PR[GP1:91,2] = PR[GP1:90,2] + -14.518;
   1:L PR[91] 10mm/sec CNT100;
   1:  PR[GP1:91,1] = PR[GP1:90,1] + 72.871;
   1:  PR[GP1:91,2] = PR[GP1:90,2] + -5.275;
   1:L PR[91] 10mm/sec CNT100;
   1:  PR[GP1:91,1] = PR[GP1:90,1] + 73.822;
   1:  PR[GP1:91,2] = PR[GP1:90,2] + -2.519;
   1:L PR[91] 10mm/sec CNT100;
   1:  PR[GP1:91,1] = PR[GP1:90,1] + 74.129;
   1:  PR[GP1:91,2] = PR[GP1:90,2] + 0.245;
   1:L PR[91] 10mm/sec CNT100;
   1:  PR[GP1:91,1] = PR[GP1:90,1] + 72.041;
   1:  PR[GP1:91,2] = PR[GP1:90,2] + 9.488;
   1:L PR[91] 10mm/sec CNT100;
   1:  PR[GP1:91,1] = PR[GP1:90,1] + 71.719;
   1:  PR[GP1:91,2] = PR[GP1:90,2] + 12.386;
   1:L PR[91] 10mm/sec CNT100;
   1:  PR[GP1:91,1] = PR[GP1:90,1] + 70.801;
   1:  PR[GP1:91,2] = PR[GP1:90,2] + 15.048;
   1:L PR[91] 10mm/sec CNT100;
   1:  PR[GP1:91,1] = PR[GP1:90,1] + 69.303;
   1:  PR[GP1:91,2] = PR[GP1:90,2] + 17.471;
   1:L PR[91] 10mm/sec CNT100;
   1:  PR[GP1:91,1] = PR[GP1:90,1] + 63.447;
   1:  PR[GP1:91,2] = PR[GP1:90,2] + 24.917;
   1:L PR[91] 10mm/sec CNT100;
   1:  PR[GP1:91,1] = PR[GP1:90,1] + 61.453;
   1:  PR[GP1:91,2] = PR[GP1:90,2] + 26.953;
   1:L PR[91] 10mm/sec CNT100;
   1:  PR[GP1:91,1] = PR[GP1:90,1] + 59.062;
   1:  PR[GP1:91,2] = PR[GP1:90,2] + 28.500;
   1:L PR[91] 10mm/sec CNT100;
   1:  PR[GP1:91,1] = PR[GP1:90,1] + 50.573;
   1:  PR[GP1:91,2] = PR[GP1:90,2] + 32.708;
   1:L PR[91] 10mm/sec CNT100;
   1:  PR[GP1:91,1] = PR[GP1:90,1] + 47.898;
   1:  PR[GP1:91,2] = PR[GP1:90,2] + 33.693;
   1:L PR[91] 10mm/sec CNT100;
   1:  PR[GP1:91,1] = PR[GP1:90,1] + 45.075;
   1:  PR[GP1:91,2] = PR[GP1:90,2] + 34.066;
   1:L PR[91] 10mm/sec CNT100;
   1:  PR[GP1:91,1] = PR[GP1:90,1] + 35.599;
   1:  PR[GP1:91,2] = PR[GP1:90,2] + 34.217;
   1:L PR[91] 10mm/sec CNT100;
   1:  PR[GP1:91,1] = PR[GP1:90,1] + 32.760;
   1:  PR[GP1:91,2] = PR[GP1:90,2] + 33.960;
   1:L PR[91] 10mm/sec CNT100;
   1:  PR[GP1:91,1] = PR[GP1:90,1] + 30.050;
   1:  PR[GP1:91,2] = PR[GP1:90,2] + 33.087;
   1:L PR[91] 10mm/sec CNT100;
   1:  PR[GP1:91,1] = PR[GP1:90,1] + 21.431;
   1:  PR[GP1:91,2] = PR[GP1:90,2] + 29.151;
   1:L PR[91] 10mm/sec CNT100;
   1:  PR[GP1:91,1] = PR[GP1:90,1] + 18.976;
   1:  PR[GP1:91,2] = PR[GP1:90,2] + 27.703;
   1:L PR[91] 10mm/sec CNT100;
   1:  PR[GP1:91,1] = PR[GP1:90,1] + 16.902;
   1:  PR[GP1:91,2] = PR[GP1:90,2] + 25.753;
   1:L PR[91] 10mm/sec CNT100;
   1:  PR[GP1:91,1] = PR[GP1:90,1] + 10.812;
   1:  PR[GP1:91,2] = PR[GP1:90,2] + 18.497;
   1:L PR[91] 10mm/sec CNT100;
   1:  PR[GP1:91,1] = PR[GP1:90,1] + 9.214;
   1:  PR[GP1:91,2] = PR[GP1:90,2] + 16.135;
   1:L PR[91] 10mm/sec CNT100;
   1:  PR[GP1:91,1] = PR[GP1:90,1] + 8.175;
   1:  PR[GP1:91,2] = PR[GP1:90,2] + 13.485;
   1:L PR[91] 10mm/sec CNT100;
   1:  PR[GP1:91,1] = PR[GP1:90,1] + 5.794;
   1:  PR[GP1:91,2] = PR[GP1:90,2] + 4.319;
   1:L PR[91] 10mm/sec CNT100;
   1:  PR[GP1:91,1] = PR[GP1:90,1] + 5.358;
   1:  PR[GP1:91,2] = PR[GP1:90,2] + 1.468;
   1:L PR[91] 10mm/sec CNT100;
   1:  PR[GP1:91,1] = PR[GP1:90,1] + 5.333;
   1:  PR[GP1:91,2] = PR[GP1:90,2] + 0.804;
   1:L PR[91] 10mm/sec CNT100;
   1:  PR[GP1:91,1] = PR[GP1:90,1] + -5.745;
   1:L PR[91] 10mm/sec CNT100;
   1:  PR[GP1:91,1] = PR[GP1:90,1] + -7.590;
   1:  PR[GP1:91,2] = PR[GP1:90,2] + 7.905;
   1:L PR[91] 10mm/sec CNT100;
   1:  PR[GP1:91,1] = PR[GP1:90,1] + -8.273;
   1:  PR[GP1:91,2] = PR[GP1:90,2] + 10.637;
   1:L PR[91] 10mm/sec CNT100;
   1:  PR[GP1:91,1] = PR[GP1:90,1] + -8.713;
   1:  PR[GP1:91,2] = PR[GP1:90,2] + 13.514;
   1:L PR[91] 10mm/sec CNT100;
   1:  PR[GP1:91,1] = PR[GP1:90,1] + -9.729;
   1:  PR[GP1:91,2] = PR[GP1:90,2] + 16.106;
   1:L PR[91] 10mm/sec CNT100;
   1:  PR[GP1:91,1] = PR[GP1:90,1] + -15.818;
   1:  PR[GP1:91,2] = PR[GP1:90,2] + 23.361;
   1:L PR[91] 10mm/sec CNT100;
   1:  PR[GP1:91,1] = PR[GP1:90,1] + -17.451;
   1:  PR[GP1:91,2] = PR[GP1:90,2] + 25.774;
   1:L PR[91] 10mm/sec CNT100;
   1:  PR[GP1:91,1] = PR[GP1:90,1] + -19.479;
   1:  PR[GP1:91,2] = PR[GP1:90,2] + 27.681;
   1:L PR[91] 10mm/sec CNT100;
   1:  PR[GP1:91,1] = PR[GP1:90,1] + -28.097;
   1:  PR[GP1:91,2] = PR[GP1:90,2] + 31.616;
   1:L PR[91] 10mm/sec CNT100;
   1:  PR[GP1:91,1] = PR[GP1:90,1] + -30.606;
   1:  PR[GP1:91,2] = PR[GP1:90,2] + 33.097;
   1:L PR[91] 10mm/sec CNT100;
   1:  PR[GP1:91,1] = PR[GP1:90,1] + -33.255;
   1:  PR[GP1:91,2] = PR[GP1:90,2] + 33.950;
   1:L PR[91] 10mm/sec CNT100;
   1:  PR[GP1:91,1] = PR[GP1:90,1] + -42.731;
   1:  PR[GP1:91,2] = PR[GP1:90,2] + 33.799;
   1:L PR[91] 10mm/sec CNT100;
   1:  PR[GP1:91,1] = PR[GP1:90,1] + -45.633;
   1:  PR[GP1:91,2] = PR[GP1:90,2] + 34.062;
   1:L PR[91] 10mm/sec CNT100;
   1:  PR[GP1:91,1] = PR[GP1:90,1] + -48.392;
   1:  PR[GP1:91,2] = PR[GP1:90,2] + 33.697;
   1:L PR[91] 10mm/sec CNT100;
   1:  PR[GP1:91,1] = PR[GP1:90,1] + -56.880;
   1:  PR[GP1:91,2] = PR[GP1:90,2] + 29.489;
   1:L PR[91] 10mm/sec CNT100;
   1:  PR[GP1:91,1] = PR[GP1:90,1] + -59.615;
   1:  PR[GP1:91,2] = PR[GP1:90,2] + 28.482;
   1:L PR[91] 10mm/sec CNT100;
   1:  PR[GP1:91,1] = PR[GP1:90,1] + -61.951;
   1:  PR[GP1:91,2] = PR[GP1:90,2] + 26.971;
   1:L PR[91] 10mm/sec CNT100;
   1:  PR[GP1:91,1] = PR[GP1:90,1] + -67.807;
   1:  PR[GP1:91,2] = PR[GP1:90,2] + 19.525;
   1:L PR[91] 10mm/sec CNT100;
   1:  PR[GP1:91,1] = PR[GP1:90,1] + -69.847;
   1:  PR[GP1:91,2] = PR[GP1:90,2] + 17.443;
   1:L PR[91] 10mm/sec CNT100;
   1:  PR[GP1:91,1] = PR[GP1:90,1] + -71.309;
   1:  PR[GP1:91,2] = PR[GP1:90,2] + 15.076;
   1:L PR[91] 10mm/sec CNT100;
   1:  PR[GP1:91,1] = PR[GP1:90,1] + -73.398;
   1:  PR[GP1:91,2] = PR[GP1:90,2] + 5.833;
   1:L PR[91] 10mm/sec CNT100;
   1:  PR[GP1:91,1] = PR[GP1:90,1] + -74.348;
   1:  PR[GP1:91,2] = PR[GP1:90,2] + 3.077;
   1:L PR[91] 10mm/sec CNT100;
   1:  PR[GP1:91,1] = PR[GP1:90,1] + -74.656;
   1:  PR[GP1:91,2] = PR[GP1:90,2] + 0.313;
   1:L PR[91] 10mm/sec CNT100;
   1:  PR[GP1:91,1] = PR[GP1:90,1] + -72.568;
   1:  PR[GP1:91,2] = PR[GP1:90,2] + -8.930;
   1:L PR[91] 10mm/sec CNT100;
   1:  PR[GP1:91,1] = PR[GP1:90,1] + -72.245;
   1:  PR[GP1:91,2] = PR[GP1:90,2] + -11.828;
   1:L PR[91] 10mm/sec CNT100;
   1:  PR[GP1:91,1] = PR[GP1:90,1] + -71.327;
   1:  PR[GP1:91,2] = PR[GP1:90,2] + -14.490;
   1:L PR[91] 10mm/sec CNT100;
   1:  PR[GP1:91,1] = PR[GP1:90,1] + -69.830;
   1:  PR[GP1:91,2] = PR[GP1:90,2] + -16.913;
   1:L PR[91] 10mm/sec CNT100;
   1:  PR[GP1:91,1] = PR[GP1:90,1] + -63.973;
   1:  PR[GP1:91,2] = PR[GP1:90,2] + -24.359;
   1:L PR[91] 10mm/sec CNT100;
   1:  PR[GP1:91,1] = PR[GP1:90,1] + -61.979;
   1:  PR[GP1:91,2] = PR[GP1:90,2] + -26.395;
   1:L PR[91] 10mm/sec CNT100;
   1:  PR[GP1:91,1] = PR[GP1:90,1] + -59.588;
   1:  PR[GP1:91,2] = PR[GP1:90,2] + -27.942;
   1:L PR[91] 10mm/sec CNT100;
   1:  PR[GP1:91,1] = PR[GP1:90,1] + -51.099;
   1:  PR[GP1:91,2] = PR[GP1:90,2] + -32.150;
   1:L PR[91] 10mm/sec CNT100;
   1:  PR[GP1:91,1] = PR[GP1:90,1] + -48.425;
   1:  PR[GP1:91,2] = PR[GP1:90,2] + -33.135;
   1:L PR[91] 10mm/sec CNT100;
   1:  PR[GP1:91,1] = PR[GP1:90,1] + -45.602;
   1:  PR[GP1:91,2] = PR[GP1:90,2] + -33.508;
   1:L PR[91] 10mm/sec CNT100;
   1:  PR[GP1:91,1] = PR[GP1:90,1] + -36.125;
   1:  PR[GP1:91,2] = PR[GP1:90,2] + -33.659;
   1:L PR[91] 10mm/sec CNT100;
   1:  PR[GP1:91,1] = PR[GP1:90,1] + -33.286;
   1:  PR[GP1:91,2] = PR[GP1:90,2] + -33.402;
   1:L PR[91] 10mm/sec CNT100;
   1:  PR[GP1:91,1] = PR[GP1:90,1] + -30.576;
   1:  PR[GP1:91,2] = PR[GP1:90,2] + -32.529;
   1:L PR[91] 10mm/sec CNT100;
   1:  PR[GP1:91,1] = PR[GP1:90,1] + -21.958;
   1:  PR[GP1:91,2] = PR[GP1:90,2] + -28.593;
   1:L PR[91] 10mm/sec CNT100;
   1:  PR[GP1:91,1] = PR[GP1:90,1] + -19.502;
   1:  PR[GP1:91,2] = PR[GP1:90,2] + -27.145;
   1:L PR[91] 10mm/sec CNT100;
   1:  PR[GP1:91,1] = PR[GP1:90,1] + -17.428;
   1:  PR[GP1:91,2] = PR[GP1:90,2] + -25.195;
   1:L PR[91] 10mm/sec CNT100;
   1:  PR[GP1:91,1] = PR[GP1:90,1] + -11.338;
   1:  PR[GP1:91,2] = PR[GP1:90,2] + -17.939;
   1:L PR[91] 10mm/sec CNT100;
   1:  PR[GP1:91,1] = PR[GP1:90,1] + -9.740;
   1:  PR[GP1:91,2] = PR[GP1:90,2] + -15.577;
   1:L PR[91] 10mm/sec CNT100;
   1:  PR[GP1:91,1] = PR[GP1:90,1] + -8.702;
   1:  PR[GP1:91,2] = PR[GP1:90,2] + -12.927;
   1:L PR[91] 10mm/sec CNT100;
   1:  PR[GP1:91,1] = PR[GP1:90,1] + -6.320;
   1:  PR[GP1:91,2] = PR[GP1:90,2] + -3.761;
   1:L PR[91] 10mm/sec CNT100;
   1:  PR[GP1:91,1] = PR[GP1:90,1] + -5.884;
   1:  PR[GP1:91,2] = PR[GP1:90,2] + -0.910;
   1:L PR[91] 10mm/sec CNT100;
   1:  PR[GP1:91,1] = PR[GP1:90,1] + -5.860;
   1:  PR[GP1:91,2] = PR[GP1:90,2] + -0.246;
   1:L PR[91] 10mm/sec CNT100;
   1:  PR[GP1:91,1] = PR[GP1:90,1] + 5.219;
   1:L PR[91] 10mm/sec CNT100;
   1:  PR[GP1:91,1] = PR[GP1:90,1] + 6.634;
   1:  PR[GP1:91,2] = PR[GP1:90,2] + -5.693;
   1:  PR[GP1:91,3] = PR[GP1:90,3] + 3.965;
   1:L PR[91] 10mm/sec CNT100;
   1:  PR[GP1:91,1] = PR[GP1:90,1] + 7.452;
   1:  PR[GP1:91,2] = PR[GP1:90,2] + -8.966;
   1:L PR[91] 10mm/sec CNT100;
   1:  PR[GP1:91,1] = PR[GP1:90,1] + 7.981;
   1:  PR[GP1:91,2] = PR[GP1:90,2] + -12.425;
   1:L PR[91] 10mm/sec CNT100;
   1:  PR[GP1:91,1] = PR[GP1:90,1] + 9.212;
   1:  PR[GP1:91,2] = PR[GP1:90,2] + -15.567;
   1:L PR[91] 10mm/sec CNT100;
   1:  PR[GP1:91,1] = PR[GP1:90,1] + 14.546;
   1:  PR[GP1:91,2] = PR[GP1:90,2] + -21.922;
   1:L PR[91] 10mm/sec CNT100;
   1:  PR[GP1:91,1] = PR[GP1:90,1] + 16.509;
   1:  PR[GP1:91,2] = PR[GP1:90,2] + -24.823;
   1:L PR[91] 10mm/sec CNT100;
   1:  PR[GP1:91,1] = PR[GP1:90,1] + 18.967;
   1:  PR[GP1:91,2] = PR[GP1:90,2] + -27.134;
   1:L PR[91] 10mm/sec CNT100;
   1:  PR[GP1:91,1] = PR[GP1:90,1] + 26.515;
   1:  PR[GP1:91,2] = PR[GP1:90,2] + -30.581;
   1:L PR[91] 10mm/sec CNT100;
   1:  PR[GP1:91,1] = PR[GP1:90,1] + 29.532;
   1:  PR[GP1:91,2] = PR[GP1:90,2] + -32.361;
   1:L PR[91] 10mm/sec CNT100;
   1:  PR[GP1:91,1] = PR[GP1:90,1] + 32.743;
   1:  PR[GP1:91,2] = PR[GP1:90,2] + -33.395;
   1:L PR[91] 10mm/sec CNT100;
   1:  PR[GP1:91,1] = PR[GP1:90,1] + 41.043;
   1:  PR[GP1:91,2] = PR[GP1:90,2] + -33.263;
   1:L PR[91] 10mm/sec CNT100;
   1:  PR[GP1:91,1] = PR[GP1:90,1] + 44.533;
   1:  PR[GP1:91,2] = PR[GP1:90,2] + -33.578;
   1:L PR[91] 10mm/sec CNT100;
   1:  PR[GP1:91,1] = PR[GP1:90,1] + 47.876;
   1:  PR[GP1:91,2] = PR[GP1:90,2] + -33.137;
   1:L PR[91] 10mm/sec CNT100;
   1:  PR[GP1:91,1] = PR[GP1:90,1] + 55.311;
   1:  PR[GP1:91,2] = PR[GP1:90,2] + -29.451;
   1:L PR[91] 10mm/sec CNT100;
   1:  PR[GP1:91,1] = PR[GP1:90,1] + 58.599;
   1:  PR[GP1:91,2] = PR[GP1:90,2] + -28.240;
   1:L PR[91] 10mm/sec CNT100;
   1:  PR[GP1:91,1] = PR[GP1:90,1] + 61.430;
   1:  PR[GP1:91,2] = PR[GP1:90,2] + -26.408;
   1:L PR[91] 10mm/sec CNT100;
   1:  PR[GP1:91,1] = PR[GP1:90,1] + 66.559;
   1:  PR[GP1:91,2] = PR[GP1:90,2] + -19.887;
   1:L PR[91] 10mm/sec CNT100;
   1:  PR[GP1:91,1] = PR[GP1:90,1] + 69.012;
   1:  PR[GP1:91,2] = PR[GP1:90,2] + -17.383;
   1:L PR[91] 10mm/sec CNT100;
   1:  PR[GP1:91,1] = PR[GP1:90,1] + 70.785;
   1:  PR[GP1:91,2] = PR[GP1:90,2] + -14.515;
   1:L PR[91] 10mm/sec CNT100;
   1:  PR[GP1:91,1] = PR[GP1:90,1] + 72.614;
   1:  PR[GP1:91,2] = PR[GP1:90,2] + -6.419;
   1:L PR[91] 10mm/sec CNT100;
   1:  PR[GP1:91,1] = PR[GP1:90,1] + 73.757;
   1:  PR[GP1:91,2] = PR[GP1:90,2] + -3.106;
   1:L PR[91] 10mm/sec CNT100;
   1:  PR[GP1:91,1] = PR[GP1:90,1] + 74.129;
   1:  PR[GP1:91,2] = PR[GP1:90,2] + 0.245;
   1:L PR[91] 10mm/sec CNT100;
   1:  PR[GP1:91,1] = PR[GP1:90,1] + 72.300;
   1:  PR[GP1:91,2] = PR[GP1:90,2] + 8.341;
   1:L PR[91] 10mm/sec CNT100;
   1:  PR[GP1:91,1] = PR[GP1:90,1] + 71.913;
   1:  PR[GP1:91,2] = PR[GP1:90,2] + 11.825;
   1:L PR[91] 10mm/sec CNT100;
   1:  PR[GP1:91,1] = PR[GP1:90,1] + 70.802;
   1:  PR[GP1:91,2] = PR[GP1:90,2] + 15.044;
   1:L PR[91] 10mm/sec CNT100;
   1:  PR[GP1:91,1] = PR[GP1:90,1] + 68.995;
   1:  PR[GP1:91,2] = PR[GP1:90,2] + 17.969;
   1:L PR[91] 10mm/sec CNT100;
   1:  PR[GP1:91,1] = PR[GP1:90,1] + 63.865;
   1:  PR[GP1:91,2] = PR[GP1:90,2] + 24.491;
   1:L PR[91] 10mm/sec CNT100;
   1:  PR[GP1:91,1] = PR[GP1:90,1] + 61.458;
   1:  PR[GP1:91,2] = PR[GP1:90,2] + 26.948;
   1:L PR[91] 10mm/sec CNT100;
   1:  PR[GP1:91,1] = PR[GP1:90,1] + 58.572;
   1:  PR[GP1:91,2] = PR[GP1:90,2] + 28.816;
   1:L PR[91] 10mm/sec CNT100;
   1:  PR[GP1:91,1] = PR[GP1:90,1] + 51.137;
   1:  PR[GP1:91,2] = PR[GP1:90,2] + 32.502;
   1:L PR[91] 10mm/sec CNT100;
   1:  PR[GP1:91,1] = PR[GP1:90,1] + 47.909;
   1:  PR[GP1:91,2] = PR[GP1:90,2] + 33.690;
   1:L PR[91] 10mm/sec CNT100;
   1:  PR[GP1:91,1] = PR[GP1:90,1] + 44.501;
   1:  PR[GP1:91,2] = PR[GP1:90,2] + 34.140;
   1:L PR[91] 10mm/sec CNT100;
   1:  PR[GP1:91,1] = PR[GP1:90,1] + 36.200;
   1:  PR[GP1:91,2] = PR[GP1:90,2] + 34.273;
   1:L PR[91] 10mm/sec CNT100;
   1:  PR[GP1:91,1] = PR[GP1:90,1] + 32.774;
   1:  PR[GP1:91,2] = PR[GP1:90,2] + 33.963;
   1:L PR[91] 10mm/sec CNT100;
   1:  PR[GP1:91,1] = PR[GP1:90,1] + 29.502;
   1:  PR[GP1:91,2] = PR[GP1:90,2] + 32.909;
   1:L PR[91] 10mm/sec CNT100;
   1:  PR[GP1:91,1] = PR[GP1:90,1] + 21.954;
   1:  PR[GP1:91,2] = PR[GP1:90,2] + 29.462;
   1:L PR[91] 10mm/sec CNT100;
   1:  PR[GP1:91,1] = PR[GP1:90,1] + 18.990;
   1:  PR[GP1:91,2] = PR[GP1:90,2] + 27.714;
   1:L PR[91] 10mm/sec CNT100;
   1:  PR[GP1:91,1] = PR[GP1:90,1] + 16.486;
   1:  PR[GP1:91,2] = PR[GP1:90,2] + 25.360;
   1:L PR[91] 10mm/sec CNT100;
   1:  PR[GP1:91,1] = PR[GP1:90,1] + 11.152;
   1:  PR[GP1:91,2] = PR[GP1:90,2] + 19.004;
   1:L PR[91] 10mm/sec CNT100;
   1:  PR[GP1:91,1] = PR[GP1:90,1] + 9.224;
   1:  PR[GP1:91,2] = PR[GP1:90,2] + 16.154;
   1:L PR[91] 10mm/sec CNT100;
   1:  PR[GP1:91,1] = PR[GP1:90,1] + 7.970;
   1:  PR[GP1:91,2] = PR[GP1:90,2] + 12.955;
   1:L PR[91] 10mm/sec CNT100;
   1:  PR[GP1:91,1] = PR[GP1:90,1] + 5.884;
   1:  PR[GP1:91,2] = PR[GP1:90,2] + 4.926;
   1:L PR[91] 10mm/sec CNT100;
   1:  PR[GP1:91,1] = PR[GP1:90,1] + 5.359;
   1:  PR[GP1:91,2] = PR[GP1:90,2] + 1.492;
   1:L PR[91] 10mm/sec CNT100;
   1:  PR[GP1:91,1] = PR[GP1:90,1] + 5.333;
   1:  PR[GP1:91,2] = PR[GP1:90,2] + 0.804;
   1:L PR[91] 10mm/sec CNT100;
   1:  PR[GP1:91,1] = PR[GP1:90,1] + -5.745;
   1:L PR[91] 10mm/sec CNT100;
   1:  PR[GP1:91,1] = PR[GP1:90,1] + -7.160;
   1:  PR[GP1:91,2] = PR[GP1:90,2] + 6.251;
   1:L PR[91] 10mm/sec CNT100;
   1:  PR[GP1:91,1] = PR[GP1:90,1] + -7.978;
   1:  PR[GP1:91,2] = PR[GP1:90,2] + 9.524;
   1:L PR[91] 10mm/sec CNT100;
   1:  PR[GP1:91,1] = PR[GP1:90,1] + -8.508;
   1:  PR[GP1:91,2] = PR[GP1:90,2] + 12.983;
   1:L PR[91] 10mm/sec CNT100;
   1:  PR[GP1:91,1] = PR[GP1:90,1] + -9.738;
   1:  PR[GP1:91,2] = PR[GP1:90,2] + 16.125;
   1:L PR[91] 10mm/sec CNT100;
   1:  PR[GP1:91,1] = PR[GP1:90,1] + -15.072;
   1:  PR[GP1:91,2] = PR[GP1:90,2] + 22.480;
   1:L PR[91] 10mm/sec CNT100;
   1:  PR[GP1:91,1] = PR[GP1:90,1] + -17.035;
   1:  PR[GP1:91,2] = PR[GP1:90,2] + 25.381;
   1:L PR[91] 10mm/sec CNT100;
   1:  PR[GP1:91,1] = PR[GP1:90,1] + -19.493;
   1:  PR[GP1:91,2] = PR[GP1:90,2] + 27.692;
   1:L PR[91] 10mm/sec CNT100;
   1:  PR[GP1:91,1] = PR[GP1:90,1] + -27.041;
   1:  PR[GP1:91,2] = PR[GP1:90,2] + 31.139;
   1:L PR[91] 10mm/sec CNT100;
   1:  PR[GP1:91,1] = PR[GP1:90,1] + -30.059;
   1:  PR[GP1:91,2] = PR[GP1:90,2] + 32.919;
   1:L PR[91] 10mm/sec CNT100;
   1:  PR[GP1:91,1] = PR[GP1:90,1] + -33.269;
   1:  PR[GP1:91,2] = PR[GP1:90,2] + 33.953;
   1:L PR[91] 10mm/sec CNT100;
   1:  PR[GP1:91,1] = PR[GP1:90,1] + -41.569;
   1:  PR[GP1:91,2] = PR[GP1:90,2] + 33.821;
   1:L PR[91] 10mm/sec CNT100;
   1:  PR[GP1:91,1] = PR[GP1:90,1] + -45.059;
   1:  PR[GP1:91,2] = PR[GP1:90,2] + 34.136;
   1:L PR[91] 10mm/sec CNT100;
   1:  PR[GP1:91,1] = PR[GP1:90,1] + -48.402;
   1:  PR[GP1:91,2] = PR[GP1:90,2] + 33.695;
   1:L PR[91] 10mm/sec CNT100;
   1:  PR[GP1:91,1] = PR[GP1:90,1] + -55.837;
   1:  PR[GP1:91,2] = PR[GP1:90,2] + 30.009;
   1:L PR[91] 10mm/sec CNT100;
   1:  PR[GP1:91,1] = PR[GP1:90,1] + -59.126;
   1:  PR[GP1:91,2] = PR[GP1:90,2] + 28.798;
   1:L PR[91] 10mm/sec CNT100;
   1:  PR[GP1:91,1] = PR[GP1:90,1] + -61.957;
   1:  PR[GP1:91,2] = PR[GP1:90,2] + 26.966;
   1:L PR[91] 10mm/sec CNT100;
   1:  PR[GP1:91,1] = PR[GP1:90,1] + -67.086;
   1:  PR[GP1:91,2] = PR[GP1:90,2] + 20.445;
   1:L PR[91] 10mm/sec CNT100;
   1:  PR[GP1:91,1] = PR[GP1:90,1] + -69.538;
   1:  PR[GP1:91,2] = PR[GP1:90,2] + 17.941;
   1:L PR[91] 10mm/sec CNT100;
   1:  PR[GP1:91,1] = PR[GP1:90,1] + -71.311;
   1:  PR[GP1:91,2] = PR[GP1:90,2] + 15.073;
   1:L PR[91] 10mm/sec CNT100;
   1:  PR[GP1:91,1] = PR[GP1:90,1] + -73.140;
   1:  PR[GP1:91,2] = PR[GP1:90,2] + 6.977;
   1:L PR[91] 10mm/sec CNT100;
   1:  PR[GP1:91,1] = PR[GP1:90,1] + -74.283;
   1:  PR[GP1:91,2] = PR[GP1:90,2] + 3.664;
   1:L PR[91] 10mm/sec CNT100;
   1:  PR[GP1:91,1] = PR[GP1:90,1] + -74.656;
   1:  PR[GP1:91,2] = PR[GP1:90,2] + 0.313;
   1:L PR[91] 10mm/sec CNT100;
   1:  PR[GP1:91,1] = PR[GP1:90,1] + -72.827;
   1:  PR[GP1:91,2] = PR[GP1:90,2] + -7.783;
   1:L PR[91] 10mm/sec CNT100;
   1:  PR[GP1:91,1] = PR[GP1:90,1] + -72.439;
   1:  PR[GP1:91,2] = PR[GP1:90,2] + -11.267;
   1:L PR[91] 10mm/sec CNT100;
   1:  PR[GP1:91,1] = PR[GP1:90,1] + -71.329;
   1:  PR[GP1:91,2] = PR[GP1:90,2] + -14.486;
   1:L PR[91] 10mm/sec CNT100;
   1:  PR[GP1:91,1] = PR[GP1:90,1] + -69.521;
   1:  PR[GP1:91,2] = PR[GP1:90,2] + -17.411;
   1:L PR[91] 10mm/sec CNT100;
   1:  PR[GP1:91,1] = PR[GP1:90,1] + -64.392;
   1:  PR[GP1:91,2] = PR[GP1:90,2] + -23.933;
   1:L PR[91] 10mm/sec CNT100;
   1:  PR[GP1:91,1] = PR[GP1:90,1] + -61.985;
   1:  PR[GP1:91,2] = PR[GP1:90,2] + -26.390;
   1:L PR[91] 10mm/sec CNT100;
   1:  PR[GP1:91,1] = PR[GP1:90,1] + -59.098;
   1:  PR[GP1:91,2] = PR[GP1:90,2] + -28.258;
   1:L PR[91] 10mm/sec CNT100;
   1:  PR[GP1:91,1] = PR[GP1:90,1] + -51.663;
   1:  PR[GP1:91,2] = PR[GP1:90,2] + -31.944;
   1:L PR[91] 10mm/sec CNT100;
   1:  PR[GP1:91,1] = PR[GP1:90,1] + -48.435;
   1:  PR[GP1:91,2] = PR[GP1:90,2] + -33.132;
   1:L PR[91] 10mm/sec CNT100;
   1:  PR[GP1:91,1] = PR[GP1:90,1] + -45.027;
   1:  PR[GP1:91,2] = PR[GP1:90,2] + -33.582;
   1:L PR[91] 10mm/sec CNT100;
   1:  PR[GP1:91,1] = PR[GP1:90,1] + -36.727;
   1:  PR[GP1:91,2] = PR[GP1:90,2] + -33.715;
   1:L PR[91] 10mm/sec CNT100;
   1:  PR[GP1:91,1] = PR[GP1:90,1] + -33.300;
   1:  PR[GP1:91,2] = PR[GP1:90,2] + -33.405;
   1:L PR[91] 10mm/sec CNT100;
   1:  PR[GP1:91,1] = PR[GP1:90,1] + -30.029;
   1:  PR[GP1:91,2] = PR[GP1:90,2] + -32.351;
   1:L PR[91] 10mm/sec CNT100;
   1:  PR[GP1:91,1] = PR[GP1:90,1] + -22.480;
   1:  PR[GP1:91,2] = PR[GP1:90,2] + -28.904;
   1:L PR[91] 10mm/sec CNT100;
   1:  PR[GP1:91,1] = PR[GP1:90,1] + -19.517;
   1:  PR[GP1:91,2] = PR[GP1:90,2] + -27.156;
   1:L PR[91] 10mm/sec CNT100;
   1:  PR[GP1:91,1] = PR[GP1:90,1] + -17.013;
   1:  PR[GP1:91,2] = PR[GP1:90,2] + -24.802;
   1:L PR[91] 10mm/sec CNT100;
   1:  PR[GP1:91,1] = PR[GP1:90,1] + -11.678;
   1:  PR[GP1:91,2] = PR[GP1:90,2] + -18.446;
   1:L PR[91] 10mm/sec CNT100;
   1:  PR[GP1:91,1] = PR[GP1:90,1] + -9.750;
   1:  PR[GP1:91,2] = PR[GP1:90,2] + -15.596;
   1:L PR[91] 10mm/sec CNT100;
   1:  PR[GP1:91,1] = PR[GP1:90,1] + -8.496;
   1:  PR[GP1:91,2] = PR[GP1:90,2] + -12.396;
   1:L PR[91] 10mm/sec CNT100;
   1:  PR[GP1:91,1] = PR[GP1:90,1] + -6.411;
   1:  PR[GP1:91,2] = PR[GP1:90,2] + -4.368;
   1:L PR[91] 10mm/sec CNT100;
   1:  PR[GP1:91,1] = PR[GP1:90,1] + -5.885;
   1:  PR[GP1:91,2] = PR[GP1:90,2] + -0.934;
   1:L PR[91] 10mm/sec CNT100;
   1:  PR[GP1:91,1] = PR[GP1:90,1] + -5.860;
   1:  PR[GP1:91,2] = PR[GP1:90,2] + -0.246;
   1:L PR[91] 10mm/sec CNT100;
   1:  PR[GP1:91,1] = PR[GP1:90,1] + 5.219;
   1:L PR[91] 10mm/sec CNT100;
   1:  PR[GP1:91,1] = PR[GP1:90,1] + 6.767;
   1:  PR[GP1:91,2] = PR[GP1:90,2] + -6.248;
   1:  PR[GP1:91,3] = PR[GP1:90,3] + 4.575;
   1:L PR[91] 10mm/sec CNT100;
   1:  PR[GP1:91,1] = PR[GP1:90,1] + 7.157;
   1:  PR[GP1:91,2] = PR[GP1:90,2] + -7.854;
   1:L PR[91] 10mm/sec CNT100;
   1:  PR[GP1:91,1] = PR[GP1:90,1] + 7.776;
   1:  PR[GP1:91,2] = PR[GP1:90,2] + -11.895;
   1:L PR[91] 10mm/sec CNT100;
   1:  PR[GP1:91,1] = PR[GP1:90,1] + 9.222;
   1:  PR[GP1:91,2] = PR[GP1:90,2] + -15.585;
   1:L PR[91] 10mm/sec CNT100;
   1:  PR[GP1:91,1] = PR[GP1:90,1] + 13.800;
   1:  PR[GP1:91,2] = PR[GP1:90,2] + -21.040;
   1:L PR[91] 10mm/sec CNT100;
   1:  PR[GP1:91,1] = PR[GP1:90,1] + 16.094;
   1:  PR[GP1:91,2] = PR[GP1:90,2] + -24.430;
   1:L PR[91] 10mm/sec CNT100;
   1:  PR[GP1:91,1] = PR[GP1:90,1] + 18.981;
   1:  PR[GP1:91,2] = PR[GP1:90,2] + -27.144;
   1:L PR[91] 10mm/sec CNT100;
   1:  PR[GP1:91,1] = PR[GP1:90,1] + 25.460;
   1:  PR[GP1:91,2] = PR[GP1:90,2] + -30.103;
   1:L PR[91] 10mm/sec CNT100;
   1:  PR[GP1:91,1] = PR[GP1:90,1] + 28.985;
   1:  PR[GP1:91,2] = PR[GP1:90,2] + -32.183;
   1:L PR[91] 10mm/sec CNT100;
   1:  PR[GP1:91,1] = PR[GP1:90,1] + 32.757;
   1:  PR[GP1:91,2] = PR[GP1:90,2] + -33.398;
   1:L PR[91] 10mm/sec CNT100;
   1:  PR[GP1:91,1] = PR[GP1:90,1] + 39.881;
   1:  PR[GP1:91,2] = PR[GP1:90,2] + -33.285;
   1:L PR[91] 10mm/sec CNT100;
   1:  PR[GP1:91,1] = PR[GP1:90,1] + 43.958;
   1:  PR[GP1:91,2] = PR[GP1:90,2] + -33.653;
   1:L PR[91] 10mm/sec CNT100;
   1:  PR[GP1:91,1] = PR[GP1:90,1] + 47.886;
   1:  PR[GP1:91,2] = PR[GP1:90,2] + -33.134;
   1:L PR[91] 10mm/sec CNT100;
   1:  PR[GP1:91,1] = PR[GP1:90,1] + 54.267;
   1:  PR[GP1:91,2] = PR[GP1:90,2] + -29.971;
   1:L PR[91] 10mm/sec CNT100;
   1:  PR[GP1:91,1] = PR[GP1:90,1] + 58.110;
   1:  PR[GP1:91,2] = PR[GP1:90,2] + -28.556;
   1:L PR[91] 10mm/sec CNT100;
   1:  PR[GP1:91,1] = PR[GP1:90,1] + 61.436;
   1:  PR[GP1:91,2] = PR[GP1:90,2] + -26.404;
   1:L PR[91] 10mm/sec CNT100;
   1:  PR[GP1:91,1] = PR[GP1:90,1] + 65.838;
   1:  PR[GP1:91,2] = PR[GP1:90,2] + -20.806;
   1:L PR[91] 10mm/sec CNT100;
   1:  PR[GP1:91,1] = PR[GP1:90,1] + 68.703;
   1:  PR[GP1:91,2] = PR[GP1:90,2] + -17.881;
   1:L PR[91] 10mm/sec CNT100;
   1:  PR[GP1:91,1] = PR[GP1:90,1] + 70.786;
   1:  PR[GP1:91,2] = PR[GP1:90,2] + -14.512;
   1:L PR[91] 10mm/sec CNT100;
   1:  PR[GP1:91,1] = PR[GP1:90,1] + 72.356;
   1:  PR[GP1:91,2] = PR[GP1:90,2] + -7.563;
   1:L PR[91] 10mm/sec CNT100;
   1:  PR[GP1:91,1] = PR[GP1:90,1] + 73.692;
   1:  PR[GP1:91,2] = PR[GP1:90,2] + -3.692;
   1:L PR[91] 10mm/sec CNT100;
   1:  PR[GP1:91,1] = PR[GP1:90,1] + 74.129;
   1:  PR[GP1:91,2] = PR[GP1:90,2] + 0.245;
   1:L PR[91] 10mm/sec CNT100;
   1:  PR[GP1:91,1] = PR[GP1:90,1] + 72.560;
   1:  PR[GP1:91,2] = PR[GP1:90,2] + 7.194;
   1:L PR[91] 10mm/sec CNT100;
   1:  PR[GP1:91,1] = PR[GP1:90,1] + 72.107;
   1:  PR[GP1:91,2] = PR[GP1:90,2] + 11.264;
   1:L PR[91] 10mm/sec CNT100;
   1:  PR[GP1:91,1] = PR[GP1:90,1] + 70.804;
   1:  PR[GP1:91,2] = PR[GP1:90,2] + 15.041;
   1:L PR[91] 10mm/sec CNT100;
   1:  PR[GP1:91,1] = PR[GP1:90,1] + 68.686;
   1:  PR[GP1:91,2] = PR[GP1:90,2] + 18.467;
   1:L PR[91] 10mm/sec CNT100;
   1:  PR[GP1:91,1] = PR[GP1:90,1] + 64.284;
   1:  PR[GP1:91,2] = PR[GP1:90,2] + 24.066;
   1:L PR[91] 10mm/sec CNT100;
   1:  PR[GP1:91,1] = PR[GP1:90,1] + 61.464;
   1:  PR[GP1:91,2] = PR[GP1:90,2] + 26.944;
   1:L PR[91] 10mm/sec CNT100;
   1:  PR[GP1:91,1] = PR[GP1:90,1] + 58.082;
   1:  PR[GP1:91,2] = PR[GP1:90,2] + 29.132;
   1:L PR[91] 10mm/sec CNT100;
   1:  PR[GP1:91,1] = PR[GP1:90,1] + 51.700;
   1:  PR[GP1:91,2] = PR[GP1:90,2] + 32.296;
   1:L PR[91] 10mm/sec CNT100;
   1:  PR[GP1:91,1] = PR[GP1:90,1] + 47.919;
   1:  PR[GP1:91,2] = PR[GP1:90,2] + 33.688;
   1:L PR[91] 10mm/sec CNT100;
   1:  PR[GP1:91,1] = PR[GP1:90,1] + 43.926;
   1:  PR[GP1:91,2] = PR[GP1:90,2] + 34.215;
   1:L PR[91] 10mm/sec CNT100;
   1:  PR[GP1:91,1] = PR[GP1:90,1] + 36.802;
   1:  PR[GP1:91,2] = PR[GP1:90,2] + 34.329;
   1:L PR[91] 10mm/sec CNT100;
   1:  PR[GP1:91,1] = PR[GP1:90,1] + 32.788;
   1:  PR[GP1:91,2] = PR[GP1:90,2] + 33.966;
   1:L PR[91] 10mm/sec CNT100;
   1:  PR[GP1:91,1] = PR[GP1:90,1] + 28.955;
   1:  PR[GP1:91,2] = PR[GP1:90,2] + 32.731;
   1:L PR[91] 10mm/sec CNT100;
   1:  PR[GP1:91,1] = PR[GP1:90,1] + 22.476;
   1:  PR[GP1:91,2] = PR[GP1:90,2] + 29.772;
   1:L PR[91] 10mm/sec CNT100;
   1:  PR[GP1:91,1] = PR[GP1:90,1] + 19.005;
   1:  PR[GP1:91,2] = PR[GP1:90,2] + 27.724;
   1:L PR[91] 10mm/sec CNT100;
   1:  PR[GP1:91,1] = PR[GP1:90,1] + 16.071;
   1:  PR[GP1:91,2] = PR[GP1:90,2] + 24.967;
   1:L PR[91] 10mm/sec CNT100;
   1:  PR[GP1:91,1] = PR[GP1:90,1] + 11.492;
   1:  PR[GP1:91,2] = PR[GP1:90,2] + 19.511;
   1:L PR[91] 10mm/sec CNT100;
   1:  PR[GP1:91,1] = PR[GP1:90,1] + 9.233;
   1:  PR[GP1:91,2] = PR[GP1:90,2] + 16.173;
   1:L PR[91] 10mm/sec CNT100;
   1:  PR[GP1:91,1] = PR[GP1:90,1] + 7.765;
   1:  PR[GP1:91,2] = PR[GP1:90,2] + 12.424;
   1:L PR[91] 10mm/sec CNT100;
   1:  PR[GP1:91,1] = PR[GP1:90,1] + 5.974;
   1:  PR[GP1:91,2] = PR[GP1:90,2] + 5.533;
   1:L PR[91] 10mm/sec CNT100;
   1:  PR[GP1:91,1] = PR[GP1:90,1] + 5.359;
   1:  PR[GP1:91,2] = PR[GP1:90,2] + 1.517;
   1:L PR[91] 10mm/sec CNT100;
   1:  PR[GP1:91,1] = PR[GP1:90,1] + 5.333;
   1:  PR[GP1:91,2] = PR[GP1:90,2] + 0.804;
   1:L PR[91] 10mm/sec CNT100;
   1:  PR[GP1:91,1] = PR[GP1:90,1] + -5.746;
   1:L PR[91] 10mm/sec CNT100;
   1:  PR[GP1:91,1] = PR[GP1:90,1] + -7.293;
   1:  PR[GP1:91,2] = PR[GP1:90,2] + 6.806;
   1:L PR[91] 10mm/sec CNT100;
   1:  PR[GP1:91,1] = PR[GP1:90,1] + -7.684;
   1:  PR[GP1:91,2] = PR[GP1:90,2] + 8.412;
   1:L PR[91] 10mm/sec CNT100;
   1:  PR[GP1:91,1] = PR[GP1:90,1] + -8.302;
   1:  PR[GP1:91,2] = PR[GP1:90,2] + 12.453;
   1:L PR[91] 10mm/sec CNT100;
   1:  PR[GP1:91,1] = PR[GP1:90,1] + -9.748;
   1:  PR[GP1:91,2] = PR[GP1:90,2] + 16.143;
   1:L PR[91] 10mm/sec CNT100;
   1:  PR[GP1:91,1] = PR[GP1:90,1] + -14.326;
   1:  PR[GP1:91,2] = PR[GP1:90,2] + 21.598;
   1:L PR[91] 10mm/sec CNT100;
   1:  PR[GP1:91,1] = PR[GP1:90,1] + -16.620;
   1:  PR[GP1:91,2] = PR[GP1:90,2] + 24.988;
   1:L PR[91] 10mm/sec CNT100;
   1:  PR[GP1:91,1] = PR[GP1:90,1] + -19.508;
   1:  PR[GP1:91,2] = PR[GP1:90,2] + 27.702;
   1:L PR[91] 10mm/sec CNT100;
   1:  PR[GP1:91,1] = PR[GP1:90,1] + -25.986;
   1:  PR[GP1:91,2] = PR[GP1:90,2] + 30.661;
   1:L PR[91] 10mm/sec CNT100;
   1:  PR[GP1:91,1] = PR[GP1:90,1] + -29.512;
   1:  PR[GP1:91,2] = PR[GP1:90,2] + 32.741;
   1:L PR[91] 10mm/sec CNT100;
   1:  PR[GP1:91,1] = PR[GP1:90,1] + -33.284;
   1:  PR[GP1:91,2] = PR[GP1:90,2] + 33.956;
   1:L PR[91] 10mm/sec CNT100;
   1:  PR[GP1:91,1] = PR[GP1:90,1] + -40.407;
   1:  PR[GP1:91,2] = PR[GP1:90,2] + 33.843;
   1:L PR[91] 10mm/sec CNT100;
   1:  PR[GP1:91,1] = PR[GP1:90,1] + -44.485;
   1:  PR[GP1:91,2] = PR[GP1:90,2] + 34.211;
   1:L PR[91] 10mm/sec CNT100;
   1:  PR[GP1:91,1] = PR[GP1:90,1] + -48.413;
   1:  PR[GP1:91,2] = PR[GP1:90,2] + 33.692;
   1:L PR[91] 10mm/sec CNT100;
   1:  PR[GP1:91,1] = PR[GP1:90,1] + -54.794;
   1:  PR[GP1:91,2] = PR[GP1:90,2] + 30.529;
   1:L PR[91] 10mm/sec CNT100;
   1:  PR[GP1:91,1] = PR[GP1:90,1] + -58.636;
   1:  PR[GP1:91,2] = PR[GP1:90,2] + 29.114;
   1:L PR[91] 10mm/sec CNT100;
   1:  PR[GP1:91,1] = PR[GP1:90,1] + -61.962;
   1:  PR[GP1:91,2] = PR[GP1:90,2] + 26.962;
   1:L PR[91] 10mm/sec CNT100;
   1:  PR[GP1:91,1] = PR[GP1:90,1] + -66.365;
   1:  PR[GP1:91,2] = PR[GP1:90,2] + 21.364;
   1:L PR[91] 10mm/sec CNT100;
   1:  PR[GP1:91,1] = PR[GP1:90,1] + -69.230;
   1:  PR[GP1:91,2] = PR[GP1:90,2] + 18.439;
   1:L PR[91] 10mm/sec CNT100;
   1:  PR[GP1:91,1] = PR[GP1:90,1] + -71.313;
   1:  PR[GP1:91,2] = PR[GP1:90,2] + 15.070;
   1:L PR[91] 10mm/sec CNT100;
   1:  PR[GP1:91,1] = PR[GP1:90,1] + -72.883;
   1:  PR[GP1:91,2] = PR[GP1:90,2] + 8.121;
   1:L PR[91] 10mm/sec CNT100;
   1:  PR[GP1:91,1] = PR[GP1:90,1] + -74.218;
   1:  PR[GP1:91,2] = PR[GP1:90,2] + 4.250;
   1:L PR[91] 10mm/sec CNT100;
   1:  PR[GP1:91,1] = PR[GP1:90,1] + -74.656;
   1:  PR[GP1:91,2] = PR[GP1:90,2] + 0.313;
   1:L PR[91] 10mm/sec CNT100;
   1:  PR[GP1:91,1] = PR[GP1:90,1] + -73.086;
   1:  PR[GP1:91,2] = PR[GP1:90,2] + -6.636;
   1:L PR[91] 10mm/sec CNT100;
   1:  PR[GP1:91,1] = PR[GP1:90,1] + -72.633;
   1:  PR[GP1:91,2] = PR[GP1:90,2] + -10.706;
   1:L PR[91] 10mm/sec CNT100;
   1:  PR[GP1:91,1] = PR[GP1:90,1] + -71.330;
   1:  PR[GP1:91,2] = PR[GP1:90,2] + -14.483;
   1:L PR[91] 10mm/sec CNT100;
   1:  PR[GP1:91,1] = PR[GP1:90,1] + -69.213;
   1:  PR[GP1:91,2] = PR[GP1:90,2] + -17.909;
   1:L PR[91] 10mm/sec CNT100;
   1:  PR[GP1:91,1] = PR[GP1:90,1] + -64.810;
   1:  PR[GP1:91,2] = PR[GP1:90,2] + -23.508;
   1:L PR[91] 10mm/sec CNT100;
   1:  PR[GP1:91,1] = PR[GP1:90,1] + -61.990;
   1:  PR[GP1:91,2] = PR[GP1:90,2] + -26.386;
   1:L PR[91] 10mm/sec CNT100;
   1:  PR[GP1:91,1] = PR[GP1:90,1] + -58.609;
   1:  PR[GP1:91,2] = PR[GP1:90,2] + -28.574;
   1:L PR[91] 10mm/sec CNT100;
   1:  PR[GP1:91,1] = PR[GP1:90,1] + -52.227;
   1:  PR[GP1:91,2] = PR[GP1:90,2] + -31.737;
   1:L PR[91] 10mm/sec CNT100;
   1:  PR[GP1:91,1] = PR[GP1:90,1] + -48.445;
   1:  PR[GP1:91,2] = PR[GP1:90,2] + -33.130;
   1:L PR[91] 10mm/sec CNT100;
   1:  PR[GP1:91,1] = PR[GP1:90,1] + -44.453;
   1:  PR[GP1:91,2] = PR[GP1:90,2] + -33.657;
   1:L PR[91] 10mm/sec CNT100;
   1:  PR[GP1:91,1] = PR[GP1:90,1] + -37.328;
   1:  PR[GP1:91,2] = PR[GP1:90,2] + -33.771;
   1:L PR[91] 10mm/sec CNT100;
   1:  PR[GP1:91,1] = PR[GP1:90,1] + -33.314;
   1:  PR[GP1:91,2] = PR[GP1:90,2] + -33.408;
   1:L PR[91] 10mm/sec CNT100;
   1:  PR[GP1:91,1] = PR[GP1:90,1] + -29.481;
   1:  PR[GP1:91,2] = PR[GP1:90,2] + -32.173;
   1:L PR[91] 10mm/sec CNT100;
   1:  PR[GP1:91,1] = PR[GP1:90,1] + -23.002;
   1:  PR[GP1:91,2] = PR[GP1:90,2] + -29.214;
   1:L PR[91] 10mm/sec CNT100;
   1:  PR[GP1:91,1] = PR[GP1:90,1] + -19.531;
   1:  PR[GP1:91,2] = PR[GP1:90,2] + -27.166;
   1:L PR[91] 10mm/sec CNT100;
   1:  PR[GP1:91,1] = PR[GP1:90,1] + -16.597;
   1:  PR[GP1:91,2] = PR[GP1:90,2] + -24.409;
   1:L PR[91] 10mm/sec CNT100;
   1:  PR[GP1:91,1] = PR[GP1:90,1] + -12.019;
   1:  PR[GP1:91,2] = PR[GP1:90,2] + -18.953;
   1:L PR[91] 10mm/sec CNT100;
   1:  PR[GP1:91,1] = PR[GP1:90,1] + -9.760;
   1:  PR[GP1:91,2] = PR[GP1:90,2] + -15.615;
   1:L PR[91] 10mm/sec CNT100;
   1:  PR[GP1:91,1] = PR[GP1:90,1] + -8.291;
   1:  PR[GP1:91,2] = PR[GP1:90,2] + -11.866;
   1:L PR[91] 10mm/sec CNT100;
   1:  PR[GP1:91,1] = PR[GP1:90,1] + -6.501;
   1:  PR[GP1:91,2] = PR[GP1:90,2] + -4.975;
   1:L PR[91] 10mm/sec CNT100;
   1:  PR[GP1:91,1] = PR[GP1:90,1] + -5.886;
   1:  PR[GP1:91,2] = PR[GP1:90,2] + -0.959;
   1:L PR[91] 10mm/sec CNT100;
   1:  PR[GP1:91,1] = PR[GP1:90,1] + -5.860;
   1:  PR[GP1:91,2] = PR[GP1:90,2] + -0.246;
   1:L PR[91] 10mm/sec CNT100;
   1:  PR[GP1:91,1] = PR[GP1:90,1] + 5.220;
   1:L PR[91] 10mm/sec CNT100;
   1:  PR[GP1:91,1] = PR[GP1:90,1] + 6.418;
   1:  PR[GP1:91,2] = PR[GP1:90,2] + -4.910;
   1:  PR[GP1:91,3] = PR[GP1:90,3] + 5.185;
   1:L PR[91] 10mm/sec CNT100;
   1:  PR[GP1:91,1] = PR[GP1:90,1] + 6.863;
   1:  PR[GP1:91,2] = PR[GP1:90,2] + -6.741;
   1:L PR[91] 10mm/sec CNT100;
   1:  PR[GP1:91,1] = PR[GP1:90,1] + 7.571;
   1:  PR[GP1:91,2] = PR[GP1:90,2] + -11.365;
   1:L PR[91] 10mm/sec CNT100;
   1:  PR[GP1:91,1] = PR[GP1:90,1] + 9.232;
   1:  PR[GP1:91,2] = PR[GP1:90,2] + -15.604;
   1:L PR[91] 10mm/sec CNT100;
   1:  PR[GP1:91,1] = PR[GP1:90,1] + 13.054;
   1:  PR[GP1:91,2] = PR[GP1:90,2] + -20.158;
   1:L PR[91] 10mm/sec CNT100;
   1:  PR[GP1:91,1] = PR[GP1:90,1] + 15.678;
   1:  PR[GP1:91,2] = PR[GP1:90,2] + -24.037;
   1:L PR[91] 10mm/sec CNT100;
   1:  PR[GP1:91,1] = PR[GP1:90,1] + 18.996;
   1:  PR[GP1:91,2] = PR[GP1:90,2] + -27.155;
   1:L PR[91] 10mm/sec CNT100;
   1:  PR[GP1:91,1] = PR[GP1:90,1] + 24.404;
   1:  PR[GP1:91,2] = PR[GP1:90,2] + -29.625;
   1:L PR[91] 10mm/sec CNT100;
   1:  PR[GP1:91,1] = PR[GP1:90,1] + 28.438;
   1:  PR[GP1:91,2] = PR[GP1:90,2] + -32.005;
   1:L PR[91] 10mm/sec CNT100;
   1:  PR[GP1:91,1] = PR[GP1:90,1] + 32.771;
   1:  PR[GP1:91,2] = PR[GP1:90,2] + -33.401;
   1:L PR[91] 10mm/sec CNT100;
   1:  PR[GP1:91,1] = PR[GP1:90,1] + 38.719;
   1:  PR[GP1:91,2] = PR[GP1:90,2] + -33.306;
   1:L PR[91] 10mm/sec CNT100;
   1:  PR[GP1:91,1] = PR[GP1:90,1] + 43.384;
   1:  PR[GP1:91,2] = PR[GP1:90,2] + -33.728;
   1:L PR[91] 10mm/sec CNT100;
   1:  PR[GP1:91,1] = PR[GP1:90,1] + 47.897;
   1:  PR[GP1:91,2] = PR[GP1:90,2] + -33.132;
   1:L PR[91] 10mm/sec CNT100;
   1:  PR[GP1:91,1] = PR[GP1:90,1] + 53.224;
   1:  PR[GP1:91,2] = PR[GP1:90,2] + -30.490;
   1:L PR[91] 10mm/sec CNT100;
   1:  PR[GP1:91,1] = PR[GP1:90,1] + 57.620;
   1:  PR[GP1:91,2] = PR[GP1:90,2] + -28.872;
   1:L PR[91] 10mm/sec CNT100;
   1:  PR[GP1:91,1] = PR[GP1:90,1] + 61.441;
   1:  PR[GP1:91,2] = PR[GP1:90,2] + -26.400;
   1:L PR[91] 10mm/sec CNT100;
   1:  PR[GP1:91,1] = PR[GP1:90,1] + 65.117;
   1:  PR[GP1:91,2] = PR[GP1:90,2] + -21.726;
   1:L PR[91] 10mm/sec CNT100;
   1:  PR[GP1:91,1] = PR[GP1:90,1] + 68.395;
   1:  PR[GP1:91,2] = PR[GP1:90,2] + -18.380;
   1:L PR[91] 10mm/sec CNT100;
   1:  PR[GP1:91,1] = PR[GP1:90,1] + 70.788;
   1:  PR[GP1:91,2] = PR[GP1:90,2] + -14.508;
   1:L PR[91] 10mm/sec CNT100;
   1:  PR[GP1:91,1] = PR[GP1:90,1] + 72.099;
   1:  PR[GP1:91,2] = PR[GP1:90,2] + -8.707;
   1:L PR[91] 10mm/sec CNT100;
   1:  PR[GP1:91,1] = PR[GP1:90,1] + 73.626;
   1:  PR[GP1:91,2] = PR[GP1:90,2] + -4.278;
   1:L PR[91] 10mm/sec CNT100;
   1:  PR[GP1:91,1] = PR[GP1:90,1] + 74.129;
   1:  PR[GP1:91,2] = PR[GP1:90,2] + 0.245;
   1:L PR[91] 10mm/sec CNT100;
   1:  PR[GP1:91,1] = PR[GP1:90,1] + 72.819;
   1:  PR[GP1:91,2] = PR[GP1:90,2] + 6.047;
   1:L PR[91] 10mm/sec CNT100;
   1:  PR[GP1:91,1] = PR[GP1:90,1] + 72.301;
   1:  PR[GP1:91,2] = PR[GP1:90,2] + 10.703;
   1:L PR[91] 10mm/sec CNT100;
   1:  PR[GP1:91,1] = PR[GP1:90,1] + 70.806;
   1:  PR[GP1:91,2] = PR[GP1:90,2] + 15.038;
   1:L PR[91] 10mm/sec CNT100;
   1:  PR[GP1:91,1] = PR[GP1:90,1] + 68.378;
   1:  PR[GP1:91,2] = PR[GP1:90,2] + 18.966;
   1:L PR[91] 10mm/sec CNT100;
   1:  PR[GP1:91,1] = PR[GP1:90,1] + 64.702;
   1:  PR[GP1:91,2] = PR[GP1:90,2] + 23.640;
   1:L PR[91] 10mm/sec CNT100;
   1:  PR[GP1:91,1] = PR[GP1:90,1] + 61.469;
   1:  PR[GP1:91,2] = PR[GP1:90,2] + 26.940;
   1:L PR[91] 10mm/sec CNT100;
   1:  PR[GP1:91,1] = PR[GP1:90,1] + 57.593;
   1:  PR[GP1:91,2] = PR[GP1:90,2] + 29.448;
   1:L PR[91] 10mm/sec CNT100;
   1:  PR[GP1:91,1] = PR[GP1:90,1] + 52.264;
   1:  PR[GP1:91,2] = PR[GP1:90,2] + 32.089;
   1:L PR[91] 10mm/sec CNT100;
   1:  PR[GP1:91,1] = PR[GP1:90,1] + 47.929;
   1:  PR[GP1:91,2] = PR[GP1:90,2] + 33.685;
   1:L PR[91] 10mm/sec CNT100;
   1:  PR[GP1:91,1] = PR[GP1:90,1] + 43.352;
   1:  PR[GP1:91,2] = PR[GP1:90,2] + 34.290;
   1:L PR[91] 10mm/sec CNT100;
   1:  PR[GP1:91,1] = PR[GP1:90,1] + 37.403;
   1:  PR[GP1:91,2] = PR[GP1:90,2] + 34.385;
   1:L PR[91] 10mm/sec CNT100;
   1:  PR[GP1:91,1] = PR[GP1:90,1] + 32.802;
   1:  PR[GP1:91,2] = PR[GP1:90,2] + 33.969;
   1:L PR[91] 10mm/sec CNT100;
   1:  PR[GP1:91,1] = PR[GP1:90,1] + 28.408;
   1:  PR[GP1:91,2] = PR[GP1:90,2] + 32.554;
   1:L PR[91] 10mm/sec CNT100;
   1:  PR[GP1:91,1] = PR[GP1:90,1] + 22.998;
   1:  PR[GP1:91,2] = PR[GP1:90,2] + 30.083;
   1:L PR[91] 10mm/sec CNT100;
   1:  PR[GP1:91,1] = PR[GP1:90,1] + 19.019;
   1:  PR[GP1:91,2] = PR[GP1:90,2] + 27.735;
   1:L PR[91] 10mm/sec CNT100;
   1:  PR[GP1:91,1] = PR[GP1:90,1] + 15.655;
   1:  PR[GP1:91,2] = PR[GP1:90,2] + 24.573;
   1:L PR[91] 10mm/sec CNT100;
   1:  PR[GP1:91,1] = PR[GP1:90,1] + 11.833;
   1:  PR[GP1:91,2] = PR[GP1:90,2] + 20.019;
   1:L PR[91] 10mm/sec CNT100;
   1:  PR[GP1:91,1] = PR[GP1:90,1] + 9.243;
   1:  PR[GP1:91,2] = PR[GP1:90,2] + 16.192;
   1:L PR[91] 10mm/sec CNT100;
   1:  PR[GP1:91,1] = PR[GP1:90,1] + 7.559;
   1:  PR[GP1:91,2] = PR[GP1:90,2] + 11.894;
   1:L PR[91] 10mm/sec CNT100;
   1:  PR[GP1:91,1] = PR[GP1:90,1] + 6.065;
   1:  PR[GP1:91,2] = PR[GP1:90,2] + 6.140;
   1:L PR[91] 10mm/sec CNT100;
   1:  PR[GP1:91,1] = PR[GP1:90,1] + 5.360;
   1:  PR[GP1:91,2] = PR[GP1:90,2] + 1.541;
   1:L PR[91] 10mm/sec CNT100;
   1:  PR[GP1:91,1] = PR[GP1:90,1] + 5.333;
   1:  PR[GP1:91,2] = PR[GP1:90,2] + 0.804;
   1:L PR[91] 10mm/sec CNT100;
   1:  PR[GP1:91,1] = PR[GP1:90,1] + -5.747;
   1:L PR[91] 10mm/sec CNT100;
   1:  PR[GP1:91,1] = PR[GP1:90,1] + -6.944;
   1:  PR[GP1:91,2] = PR[GP1:90,2] + 5.468;
   1:L PR[91] 10mm/sec CNT100;
   1:  PR[GP1:91,1] = PR[GP1:90,1] + -7.389;
   1:  PR[GP1:91,2] = PR[GP1:90,2] + 7.299;
   1:L PR[91] 10mm/sec CNT100;
   1:  PR[GP1:91,1] = PR[GP1:90,1] + -8.097;
   1:  PR[GP1:91,2] = PR[GP1:90,2] + 11.923;
   1:L PR[91] 10mm/sec CNT100;
   1:  PR[GP1:91,1] = PR[GP1:90,1] + -9.758;
   1:  PR[GP1:91,2] = PR[GP1:90,2] + 16.162;
   1:L PR[91] 10mm/sec CNT100;
   1:  PR[GP1:91,1] = PR[GP1:90,1] + -13.580;
   1:  PR[GP1:91,2] = PR[GP1:90,2] + 20.716;
   1:L PR[91] 10mm/sec CNT100;
   1:  PR[GP1:91,1] = PR[GP1:90,1] + -16.204;
   1:  PR[GP1:91,2] = PR[GP1:90,2] + 24.595;
   1:L PR[91] 10mm/sec CNT100;
   1:  PR[GP1:91,1] = PR[GP1:90,1] + -19.522;
   1:  PR[GP1:91,2] = PR[GP1:90,2] + 27.713;
   1:L PR[91] 10mm/sec CNT100;
   1:  PR[GP1:91,1] = PR[GP1:90,1] + -24.931;
   1:  PR[GP1:91,2] = PR[GP1:90,2] + 30.183;
   1:L PR[91] 10mm/sec CNT100;
   1:  PR[GP1:91,1] = PR[GP1:90,1] + -28.964;
   1:  PR[GP1:91,2] = PR[GP1:90,2] + 32.563;
   1:L PR[91] 10mm/sec CNT100;
   1:  PR[GP1:91,1] = PR[GP1:90,1] + -33.298;
   1:  PR[GP1:91,2] = PR[GP1:90,2] + 33.959;
   1:L PR[91] 10mm/sec CNT100;
   1:  PR[GP1:91,1] = PR[GP1:90,1] + -39.246;
   1:  PR[GP1:91,2] = PR[GP1:90,2] + 33.864;
   1:L PR[91] 10mm/sec CNT100;
   1:  PR[GP1:91,1] = PR[GP1:90,1] + -43.910;
   1:  PR[GP1:91,2] = PR[GP1:90,2] + 34.286;
   1:L PR[91] 10mm/sec CNT100;
   1:  PR[GP1:91,1] = PR[GP1:90,1] + -48.423;
   1:  PR[GP1:91,2] = PR[GP1:90,2] + 33.690;
   1:L PR[91] 10mm/sec CNT100;
   1:  PR[GP1:91,1] = PR[GP1:90,1] + -53.751;
   1:  PR[GP1:91,2] = PR[GP1:90,2] + 31.048;
   1:L PR[91] 10mm/sec CNT100;
   1:  PR[GP1:91,1] = PR[GP1:90,1] + -58.146;
   1:  PR[GP1:91,2] = PR[GP1:90,2] + 29.430;
   1:L PR[91] 10mm/sec CNT100;
   1:  PR[GP1:91,1] = PR[GP1:90,1] + -61.968;
   1:  PR[GP1:91,2] = PR[GP1:90,2] + 26.958;
   1:L PR[91] 10mm/sec CNT100;
   1:  PR[GP1:91,1] = PR[GP1:90,1] + -65.643;
   1:  PR[GP1:91,2] = PR[GP1:90,2] + 22.284;
   1:L PR[91] 10mm/sec CNT100;
   1:  PR[GP1:91,1] = PR[GP1:90,1] + -68.921;
   1:  PR[GP1:91,2] = PR[GP1:90,2] + 18.938;
   1:L PR[91] 10mm/sec CNT100;
   1:  PR[GP1:91,1] = PR[GP1:90,1] + -71.314;
   1:  PR[GP1:91,2] = PR[GP1:90,2] + 15.066;
   1:L PR[91] 10mm/sec CNT100;
   1:  PR[GP1:91,1] = PR[GP1:90,1] + -72.625;
   1:  PR[GP1:91,2] = PR[GP1:90,2] + 9.265;
   1:L PR[91] 10mm/sec CNT100;
   1:  PR[GP1:91,1] = PR[GP1:90,1] + -74.153;
   1:  PR[GP1:91,2] = PR[GP1:90,2] + 4.836;
   1:L PR[91] 10mm/sec CNT100;
   1:  PR[GP1:91,1] = PR[GP1:90,1] + -74.656;
   1:  PR[GP1:91,2] = PR[GP1:90,2] + 0.313;
   1:L PR[91] 10mm/sec CNT100;
   1:  PR[GP1:91,1] = PR[GP1:90,1] + -73.345;
   1:  PR[GP1:91,2] = PR[GP1:90,2] + -5.489;
   1:L PR[91] 10mm/sec CNT100;
   1:  PR[GP1:91,1] = PR[GP1:90,1] + -72.827;
   1:  PR[GP1:91,2] = PR[GP1:90,2] + -10.145;
   1:L PR[91] 10mm/sec CNT100;
   1:  PR[GP1:91,1] = PR[GP1:90,1] + -71.332;
   1:  PR[GP1:91,2] = PR[GP1:90,2] + -14.480;
   1:L PR[91] 10mm/sec CNT100;
   1:  PR[GP1:91,1] = PR[GP1:90,1] + -68.904;
   1:  PR[GP1:91,2] = PR[GP1:90,2] + -18.408;
   1:L PR[91] 10mm/sec CNT100;
   1:  PR[GP1:91,1] = PR[GP1:90,1] + -65.228;
   1:  PR[GP1:91,2] = PR[GP1:90,2] + -23.082;
   1:L PR[91] 10mm/sec CNT100;
   1:  PR[GP1:91,1] = PR[GP1:90,1] + -61.996;
   1:  PR[GP1:91,2] = PR[GP1:90,2] + -26.381;
   1:L PR[91] 10mm/sec CNT100;
   1:  PR[GP1:91,1] = PR[GP1:90,1] + -58.119;
   1:  PR[GP1:91,2] = PR[GP1:90,2] + -28.890;
   1:L PR[91] 10mm/sec CNT100;
   1:  PR[GP1:91,1] = PR[GP1:90,1] + -52.791;
   1:  PR[GP1:91,2] = PR[GP1:90,2] + -31.531;
   1:L PR[91] 10mm/sec CNT100;
   1:  PR[GP1:91,1] = PR[GP1:90,1] + -48.456;
   1:  PR[GP1:91,2] = PR[GP1:90,2] + -33.127;
   1:L PR[91] 10mm/sec CNT100;
   1:  PR[GP1:91,1] = PR[GP1:90,1] + -43.878;
   1:  PR[GP1:91,2] = PR[GP1:90,2] + -33.732;
   1:L PR[91] 10mm/sec CNT100;
   1:  PR[GP1:91,1] = PR[GP1:90,1] + -37.930;
   1:  PR[GP1:91,2] = PR[GP1:90,2] + -33.827;
   1:L PR[91] 10mm/sec CNT100;
   1:  PR[GP1:91,1] = PR[GP1:90,1] + -33.329;
   1:  PR[GP1:91,2] = PR[GP1:90,2] + -33.411;
   1:L PR[91] 10mm/sec CNT100;
   1:  PR[GP1:91,1] = PR[GP1:90,1] + -28.934;
   1:  PR[GP1:91,2] = PR[GP1:90,2] + -31.995;
   1:L PR[91] 10mm/sec CNT100;
   1:  PR[GP1:91,1] = PR[GP1:90,1] + -23.525;
   1:  PR[GP1:91,2] = PR[GP1:90,2] + -29.525;
   1:L PR[91] 10mm/sec CNT100;
   1:  PR[GP1:91,1] = PR[GP1:90,1] + -19.545;
   1:  PR[GP1:91,2] = PR[GP1:90,2] + -27.177;
   1:L PR[91] 10mm/sec CNT100;
   1:  PR[GP1:91,1] = PR[GP1:90,1] + -16.182;
   1:  PR[GP1:91,2] = PR[GP1:90,2] + -24.015;
   1:L PR[91] 10mm/sec CNT100;
   1:  PR[GP1:91,1] = PR[GP1:90,1] + -12.359;
   1:  PR[GP1:91,2] = PR[GP1:90,2] + -19.461;
   1:L PR[91] 10mm/sec CNT100;
   1:  PR[GP1:91,1] = PR[GP1:90,1] + -9.770;
   1:  PR[GP1:91,2] = PR[GP1:90,2] + -15.634;
   1:L PR[91] 10mm/sec CNT100;
   1:  PR[GP1:91,1] = PR[GP1:90,1] + -8.086;
   1:  PR[GP1:91,2] = PR[GP1:90,2] + -11.336;
   1:L PR[91] 10mm/sec CNT100;
   1:  PR[GP1:91,1] = PR[GP1:90,1] + -6.591;
   1:  PR[GP1:91,2] = PR[GP1:90,2] + -5.582;
   1:L PR[91] 10mm/sec CNT100;
   1:  PR[GP1:91,1] = PR[GP1:90,1] + -5.887;
   1:  PR[GP1:91,2] = PR[GP1:90,2] + -0.983;
   1:L PR[91] 10mm/sec CNT100;
   1:  PR[GP1:91,1] = PR[GP1:90,1] + -5.860;
   1:  PR[GP1:91,2] = PR[GP1:90,2] + -0.246;
   1:L PR[91] 10mm/sec CNT100;
   1:  PR[GP1:91,1] = PR[GP1:90,1] + 5.220;
   1:L PR[91] 10mm/sec CNT100;
   1:  PR[GP1:91,1] = PR[GP1:90,1] + 6.068;
   1:  PR[GP1:91,2] = PR[GP1:90,2] + -3.572;
   1:  PR[GP1:91,3] = PR[GP1:90,3] + 5.795;
   1:L PR[91] 10mm/sec CNT100;
   1:  PR[GP1:91,1] = PR[GP1:90,1] + 6.568;
   1:  PR[GP1:91,2] = PR[GP1:90,2] + -5.627;
   1:L PR[91] 10mm/sec CNT100;
   1:  PR[GP1:91,1] = PR[GP1:90,1] + 7.365;
   1:  PR[GP1:91,2] = PR[GP1:90,2] + -10.834;
   1:L PR[91] 10mm/sec CNT100;
   1:  PR[GP1:91,1] = PR[GP1:90,1] + 9.241;
   1:  PR[GP1:91,2] = PR[GP1:90,2] + -15.623;
   1:L PR[91] 10mm/sec CNT100;
   1:  PR[GP1:91,1] = PR[GP1:90,1] + 12.308;
   1:  PR[GP1:91,2] = PR[GP1:90,2] + -19.277;
   1:L PR[91] 10mm/sec CNT100;
   1:  PR[GP1:91,1] = PR[GP1:90,1] + 15.263;
   1:  PR[GP1:91,2] = PR[GP1:90,2] + -23.644;
   1:L PR[91] 10mm/sec CNT100;
   1:  PR[GP1:91,1] = PR[GP1:90,1] + 19.010;
   1:  PR[GP1:91,2] = PR[GP1:90,2] + -27.166;
   1:L PR[91] 10mm/sec CNT100;
   1:  PR[GP1:91,1] = PR[GP1:90,1] + 23.349;
   1:  PR[GP1:91,2] = PR[GP1:90,2] + -29.148;
   1:L PR[91] 10mm/sec CNT100;
   1:  PR[GP1:91,1] = PR[GP1:90,1] + 27.891;
   1:  PR[GP1:91,2] = PR[GP1:90,2] + -31.827;
   1:L PR[91] 10mm/sec CNT100;
   1:  PR[GP1:91,1] = PR[GP1:90,1] + 32.785;
   1:  PR[GP1:91,2] = PR[GP1:90,2] + -33.404;
   1:L PR[91] 10mm/sec CNT100;
   1:  PR[GP1:91,1] = PR[GP1:90,1] + 37.557;
   1:  PR[GP1:91,2] = PR[GP1:90,2] + -33.328;
   1:L PR[91] 10mm/sec CNT100;
   1:  PR[GP1:91,1] = PR[GP1:90,1] + 42.809;
   1:  PR[GP1:91,2] = PR[GP1:90,2] + -33.802;
   1:L PR[91] 10mm/sec CNT100;
   1:  PR[GP1:91,1] = PR[GP1:90,1] + 47.907;
   1:  PR[GP1:91,2] = PR[GP1:90,2] + -33.129;
   1:L PR[91] 10mm/sec CNT100;
   1:  PR[GP1:91,1] = PR[GP1:90,1] + 52.181;
   1:  PR[GP1:91,2] = PR[GP1:90,2] + -31.010;
   1:L PR[91] 10mm/sec CNT100;
   1:  PR[GP1:91,1] = PR[GP1:90,1] + 57.130;
   1:  PR[GP1:91,2] = PR[GP1:90,2] + -29.188;
   1:L PR[91] 10mm/sec CNT100;
   1:  PR[GP1:91,1] = PR[GP1:90,1] + 61.447;
   1:  PR[GP1:91,2] = PR[GP1:90,2] + -26.395;
   1:L PR[91] 10mm/sec CNT100;
   1:  PR[GP1:91,1] = PR[GP1:90,1] + 64.396;
   1:  PR[GP1:91,2] = PR[GP1:90,2] + -22.646;
   1:L PR[91] 10mm/sec CNT100;
   1:  PR[GP1:91,1] = PR[GP1:90,1] + 68.087;
   1:  PR[GP1:91,2] = PR[GP1:90,2] + -18.878;
   1:L PR[91] 10mm/sec CNT100;
   1:  PR[GP1:91,1] = PR[GP1:90,1] + 70.790;
   1:  PR[GP1:91,2] = PR[GP1:90,2] + -14.505;
   1:L PR[91] 10mm/sec CNT100;
   1:  PR[GP1:91,1] = PR[GP1:90,1] + 71.841;
   1:  PR[GP1:91,2] = PR[GP1:90,2] + -9.850;
   1:L PR[91] 10mm/sec CNT100;
   1:  PR[GP1:91,1] = PR[GP1:90,1] + 73.561;
   1:  PR[GP1:91,2] = PR[GP1:90,2] + -4.864;
   1:L PR[91] 10mm/sec CNT100;
   1:  PR[GP1:91,1] = PR[GP1:90,1] + 74.129;
   1:  PR[GP1:91,2] = PR[GP1:90,2] + 0.245;
   1:L PR[91] 10mm/sec CNT100;
   1:  PR[GP1:91,1] = PR[GP1:90,1] + 73.078;
   1:  PR[GP1:91,2] = PR[GP1:90,2] + 4.900;
   1:L PR[91] 10mm/sec CNT100;
   1:  PR[GP1:91,1] = PR[GP1:90,1] + 72.495;
   1:  PR[GP1:91,2] = PR[GP1:90,2] + 10.142;
   1:L PR[91] 10mm/sec CNT100;
   1:  PR[GP1:91,1] = PR[GP1:90,1] + 70.807;
   1:  PR[GP1:91,2] = PR[GP1:90,2] + 15.034;
   1:L PR[91] 10mm/sec CNT100;
   1:  PR[GP1:91,1] = PR[GP1:90,1] + 68.069;
   1:  PR[GP1:91,2] = PR[GP1:90,2] + 19.464;
   1:L PR[91] 10mm/sec CNT100;
   1:  PR[GP1:91,1] = PR[GP1:90,1] + 65.120;
   1:  PR[GP1:91,2] = PR[GP1:90,2] + 23.214;
   1:L PR[91] 10mm/sec CNT100;
   1:  PR[GP1:91,1] = PR[GP1:90,1] + 61.475;
   1:  PR[GP1:91,2] = PR[GP1:90,2] + 26.935;
   1:L PR[91] 10mm/sec CNT100;
   1:  PR[GP1:91,1] = PR[GP1:90,1] + 57.103;
   1:  PR[GP1:91,2] = PR[GP1:90,2] + 29.764;
   1:L PR[91] 10mm/sec CNT100;
   1:  PR[GP1:91,1] = PR[GP1:90,1] + 52.828;
   1:  PR[GP1:91,2] = PR[GP1:90,2] + 31.883;
   1:L PR[91] 10mm/sec CNT100;
   1:  PR[GP1:91,1] = PR[GP1:90,1] + 47.939;
   1:  PR[GP1:91,2] = PR[GP1:90,2] + 33.683;
   1:L PR[91] 10mm/sec CNT100;
   1:  PR[GP1:91,1] = PR[GP1:90,1] + 42.777;
   1:  PR[GP1:91,2] = PR[GP1:90,2] + 34.365;
   1:L PR[91] 10mm/sec CNT100;
   1:  PR[GP1:91,1] = PR[GP1:90,1] + 38.005;
   1:  PR[GP1:91,2] = PR[GP1:90,2] + 34.441;
   1:L PR[91] 10mm/sec CNT100;
   1:  PR[GP1:91,1] = PR[GP1:90,1] + 32.816;
   1:  PR[GP1:91,2] = PR[GP1:90,2] + 33.972;
   1:L PR[91] 10mm/sec CNT100;
   1:  PR[GP1:91,1] = PR[GP1:90,1] + 27.861;
   1:  PR[GP1:91,2] = PR[GP1:90,2] + 32.376;
   1:L PR[91] 10mm/sec CNT100;
   1:  PR[GP1:91,1] = PR[GP1:90,1] + 23.520;
   1:  PR[GP1:91,2] = PR[GP1:90,2] + 30.394;
   1:L PR[91] 10mm/sec CNT100;
   1:  PR[GP1:91,1] = PR[GP1:90,1] + 19.033;
   1:  PR[GP1:91,2] = PR[GP1:90,2] + 27.746;
   1:L PR[91] 10mm/sec CNT100;
   1:  PR[GP1:91,1] = PR[GP1:90,1] + 15.240;
   1:  PR[GP1:91,2] = PR[GP1:90,2] + 24.180;
   1:L PR[91] 10mm/sec CNT100;
   1:  PR[GP1:91,1] = PR[GP1:90,1] + 12.173;
   1:  PR[GP1:91,2] = PR[GP1:90,2] + 20.526;
   1:L PR[91] 10mm/sec CNT100;
   1:  PR[GP1:91,1] = PR[GP1:90,1] + 9.253;
   1:  PR[GP1:91,2] = PR[GP1:90,2] + 16.211;
   1:L PR[91] 10mm/sec CNT100;
   1:  PR[GP1:91,1] = PR[GP1:90,1] + 7.354;
   1:  PR[GP1:91,2] = PR[GP1:90,2] + 11.364;
   1:L PR[91] 10mm/sec CNT100;
   1:  PR[GP1:91,1] = PR[GP1:90,1] + 6.155;
   1:  PR[GP1:91,2] = PR[GP1:90,2] + 6.747;
   1:L PR[91] 10mm/sec CNT100;
   1:  PR[GP1:91,1] = PR[GP1:90,1] + 5.361;
   1:  PR[GP1:91,2] = PR[GP1:90,2] + 1.565;
   1:L PR[91] 10mm/sec CNT100;
   1:  PR[GP1:91,1] = PR[GP1:90,1] + 5.333;
   1:  PR[GP1:91,2] = PR[GP1:90,2] + 0.804;
   1:L PR[91] 10mm/sec CNT100;
   1:  PR[GP1:91,1] = PR[GP1:90,1] + -5.748;
   1:L PR[91] 10mm/sec CNT100;
   1:  PR[GP1:91,1] = PR[GP1:90,1] + -6.595;
   1:  PR[GP1:91,2] = PR[GP1:90,2] + 4.130;
   1:L PR[91] 10mm/sec CNT100;
   1:  PR[GP1:91,1] = PR[GP1:90,1] + -7.094;
   1:  PR[GP1:91,2] = PR[GP1:90,2] + 6.186;
   1:L PR[91] 10mm/sec CNT100;
   1:  PR[GP1:91,1] = PR[GP1:90,1] + -7.892;
   1:  PR[GP1:91,2] = PR[GP1:90,2] + 11.392;
   1:L PR[91] 10mm/sec CNT100;
   1:  PR[GP1:91,1] = PR[GP1:90,1] + -9.768;
   1:  PR[GP1:91,2] = PR[GP1:90,2] + 16.181;
   1:L PR[91] 10mm/sec CNT100;
   1:  PR[GP1:91,1] = PR[GP1:90,1] + -12.834;
   1:  PR[GP1:91,2] = PR[GP1:90,2] + 19.835;
   1:L PR[91] 10mm/sec CNT100;
   1:  PR[GP1:91,1] = PR[GP1:90,1] + -15.789;
   1:  PR[GP1:91,2] = PR[GP1:90,2] + 24.202;
   1:L PR[91] 10mm/sec CNT100;
   1:  PR[GP1:91,1] = PR[GP1:90,1] + -19.536;
   1:  PR[GP1:91,2] = PR[GP1:90,2] + 27.724;
   1:L PR[91] 10mm/sec CNT100;
   1:  PR[GP1:91,1] = PR[GP1:90,1] + -23.876;
   1:  PR[GP1:91,2] = PR[GP1:90,2] + 29.706;
   1:L PR[91] 10mm/sec CNT100;
   1:  PR[GP1:91,1] = PR[GP1:90,1] + -28.417;
   1:  PR[GP1:91,2] = PR[GP1:90,2] + 32.385;
   1:L PR[91] 10mm/sec CNT100;
   1:  PR[GP1:91,1] = PR[GP1:90,1] + -33.312;
   1:  PR[GP1:91,2] = PR[GP1:90,2] + 33.962;
   1:L PR[91] 10mm/sec CNT100;
   1:  PR[GP1:91,1] = PR[GP1:90,1] + -38.084;
   1:  PR[GP1:91,2] = PR[GP1:90,2] + 33.886;
   1:L PR[91] 10mm/sec CNT100;
   1:  PR[GP1:91,1] = PR[GP1:90,1] + -43.336;
   1:  PR[GP1:91,2] = PR[GP1:90,2] + 34.360;
   1:L PR[91] 10mm/sec CNT100;
   1:  PR[GP1:91,1] = PR[GP1:90,1] + -48.433;
   1:  PR[GP1:91,2] = PR[GP1:90,2] + 33.687;
   1:L PR[91] 10mm/sec CNT100;
   1:  PR[GP1:91,1] = PR[GP1:90,1] + -52.708;
   1:  PR[GP1:91,2] = PR[GP1:90,2] + 31.568;
   1:L PR[91] 10mm/sec CNT100;
   1:  PR[GP1:91,1] = PR[GP1:90,1] + -57.657;
   1:  PR[GP1:91,2] = PR[GP1:90,2] + 29.746;
   1:L PR[91] 10mm/sec CNT100;
   1:  PR[GP1:91,1] = PR[GP1:90,1] + -61.973;
   1:  PR[GP1:91,2] = PR[GP1:90,2] + 26.953;
   1:L PR[91] 10mm/sec CNT100;
   1:  PR[GP1:91,1] = PR[GP1:90,1] + -64.922;
   1:  PR[GP1:91,2] = PR[GP1:90,2] + 23.204;
   1:L PR[91] 10mm/sec CNT100;
   1:  PR[GP1:91,1] = PR[GP1:90,1] + -68.613;
   1:  PR[GP1:91,2] = PR[GP1:90,2] + 19.436;
   1:L PR[91] 10mm/sec CNT100;
   1:  PR[GP1:91,1] = PR[GP1:90,1] + -71.316;
   1:  PR[GP1:91,2] = PR[GP1:90,2] + 15.063;
   1:L PR[91] 10mm/sec CNT100;
   1:  PR[GP1:91,1] = PR[GP1:90,1] + -72.368;
   1:  PR[GP1:91,2] = PR[GP1:90,2] + 10.408;
   1:L PR[91] 10mm/sec CNT100;
   1:  PR[GP1:91,1] = PR[GP1:90,1] + -74.088;
   1:  PR[GP1:91,2] = PR[GP1:90,2] + 5.422;
   1:L PR[91] 10mm/sec CNT100;
   1:  PR[GP1:91,1] = PR[GP1:90,1] + -74.656;
   1:  PR[GP1:91,2] = PR[GP1:90,2] + 0.313;
   1:L PR[91] 10mm/sec CNT100;
   1:  PR[GP1:91,1] = PR[GP1:90,1] + -73.604;
   1:  PR[GP1:91,2] = PR[GP1:90,2] + -4.342;
   1:L PR[91] 10mm/sec CNT100;
   1:  PR[GP1:91,1] = PR[GP1:90,1] + -73.021;
   1:  PR[GP1:91,2] = PR[GP1:90,2] + -9.584;
   1:L PR[91] 10mm/sec CNT100;
   1:  PR[GP1:91,1] = PR[GP1:90,1] + -71.334;
   1:  PR[GP1:91,2] = PR[GP1:90,2] + -14.476;
   1:L PR[91] 10mm/sec CNT100;
   1:  PR[GP1:91,1] = PR[GP1:90,1] + -68.596;
   1:  PR[GP1:91,2] = PR[GP1:90,2] + -18.906;
   1:L PR[91] 10mm/sec CNT100;
   1:  PR[GP1:91,1] = PR[GP1:90,1] + -65.646;
   1:  PR[GP1:91,2] = PR[GP1:90,2] + -22.656;
   1:L PR[91] 10mm/sec CNT100;
   1:  PR[GP1:91,1] = PR[GP1:90,1] + -62.001;
   1:  PR[GP1:91,2] = PR[GP1:90,2] + -26.377;
   1:L PR[91] 10mm/sec CNT100;
   1:  PR[GP1:91,1] = PR[GP1:90,1] + -57.629;
   1:  PR[GP1:91,2] = PR[GP1:90,2] + -29.206;
   1:L PR[91] 10mm/sec CNT100;
   1:  PR[GP1:91,1] = PR[GP1:90,1] + -53.354;
   1:  PR[GP1:91,2] = PR[GP1:90,2] + -31.325;
   1:L PR[91] 10mm/sec CNT100;
   1:  PR[GP1:91,1] = PR[GP1:90,1] + -48.466;
   1:  PR[GP1:91,2] = PR[GP1:90,2] + -33.125;
   1:L PR[91] 10mm/sec CNT100;
   1:  PR[GP1:91,1] = PR[GP1:90,1] + -43.304;
   1:  PR[GP1:91,2] = PR[GP1:90,2] + -33.807;
   1:L PR[91] 10mm/sec CNT100;
   1:  PR[GP1:91,1] = PR[GP1:90,1] + -38.531;
   1:  PR[GP1:91,2] = PR[GP1:90,2] + -33.883;
   1:L PR[91] 10mm/sec CNT100;
   1:  PR[GP1:91,1] = PR[GP1:90,1] + -33.343;
   1:  PR[GP1:91,2] = PR[GP1:90,2] + -33.414;
   1:L PR[91] 10mm/sec CNT100;
   1:  PR[GP1:91,1] = PR[GP1:90,1] + -28.387;
   1:  PR[GP1:91,2] = PR[GP1:90,2] + -31.818;
   1:L PR[91] 10mm/sec CNT100;
   1:  PR[GP1:91,1] = PR[GP1:90,1] + -24.047;
   1:  PR[GP1:91,2] = PR[GP1:90,2] + -29.835;
   1:L PR[91] 10mm/sec CNT100;
   1:  PR[GP1:91,1] = PR[GP1:90,1] + -19.559;
   1:  PR[GP1:91,2] = PR[GP1:90,2] + -27.188;
   1:L PR[91] 10mm/sec CNT100;
   1:  PR[GP1:91,1] = PR[GP1:90,1] + -15.766;
   1:  PR[GP1:91,2] = PR[GP1:90,2] + -23.622;
   1:L PR[91] 10mm/sec CNT100;
   1:  PR[GP1:91,1] = PR[GP1:90,1] + -12.699;
   1:  PR[GP1:91,2] = PR[GP1:90,2] + -19.968;
   1:L PR[91] 10mm/sec CNT100;
   1:  PR[GP1:91,1] = PR[GP1:90,1] + -9.779;
   1:  PR[GP1:91,2] = PR[GP1:90,2] + -15.653;
   1:L PR[91] 10mm/sec CNT100;
   1:  PR[GP1:91,1] = PR[GP1:90,1] + -7.880;
   1:  PR[GP1:91,2] = PR[GP1:90,2] + -10.805;
   1:L PR[91] 10mm/sec CNT100;
   1:  PR[GP1:91,1] = PR[GP1:90,1] + -6.681;
   1:  PR[GP1:91,2] = PR[GP1:90,2] + -6.189;
   1:L PR[91] 10mm/sec CNT100;
   1:  PR[GP1:91,1] = PR[GP1:90,1] + -5.888;
   1:  PR[GP1:91,2] = PR[GP1:90,2] + -1.007;
   1:L PR[91] 10mm/sec CNT100;
   1:  PR[GP1:91,1] = PR[GP1:90,1] + -5.860;
   1:  PR[GP1:91,2] = PR[GP1:90,2] + -0.246;
   1:L PR[91] 10mm/sec CNT100;
   1:  PR[GP1:91,1] = PR[GP1:90,1] + 5.221;
   1:L PR[91] 10mm/sec CNT100;
   1:  PR[GP1:91,1] = PR[GP1:90,1] + 5.719;
   1:  PR[GP1:91,2] = PR[GP1:90,2] + -2.233;
   1:  PR[GP1:91,3] = PR[GP1:90,3] + 6.405;
   1:L PR[91] 10mm/sec CNT100;
   1:  PR[GP1:91,1] = PR[GP1:90,1] + 6.273;
   1:  PR[GP1:91,2] = PR[GP1:90,2] + -4.514;
   1:L PR[91] 10mm/sec CNT100;
   1:  PR[GP1:91,1] = PR[GP1:90,1] + 7.160;
   1:  PR[GP1:91,2] = PR[GP1:90,2] + -10.304;
   1:L PR[91] 10mm/sec CNT100;
   1:  PR[GP1:91,1] = PR[GP1:90,1] + 9.251;
   1:  PR[GP1:91,2] = PR[GP1:90,2] + -15.642;
   1:L PR[91] 10mm/sec CNT100;
   1:  PR[GP1:91,1] = PR[GP1:90,1] + 11.562;
   1:  PR[GP1:91,2] = PR[GP1:90,2] + -18.395;
   1:L PR[91] 10mm/sec CNT100;
   1:  PR[GP1:91,1] = PR[GP1:90,1] + 14.847;
   1:  PR[GP1:91,2] = PR[GP1:90,2] + -23.251;
   1:L PR[91] 10mm/sec CNT100;
   1:  PR[GP1:91,1] = PR[GP1:90,1] + 19.024;
   1:  PR[GP1:91,2] = PR[GP1:90,2] + -27.177;
   1:L PR[91] 10mm/sec CNT100;
   1:  PR[GP1:91,1] = PR[GP1:90,1] + 22.294;
   1:  PR[GP1:91,2] = PR[GP1:90,2] + -28.670;
   1:L PR[91] 10mm/sec CNT100;
   1:  PR[GP1:91,1] = PR[GP1:90,1] + 27.343;
   1:  PR[GP1:91,2] = PR[GP1:90,2] + -31.649;
   1:L PR[91] 10mm/sec CNT100;
   1:  PR[GP1:91,1] = PR[GP1:90,1] + 32.800;
   1:  PR[GP1:91,2] = PR[GP1:90,2] + -33.407;
   1:L PR[91] 10mm/sec CNT100;
   1:  PR[GP1:91,1] = PR[GP1:90,1] + 36.395;
   1:  PR[GP1:91,2] = PR[GP1:90,2] + -33.349;
   1:L PR[91] 10mm/sec CNT100;
   1:  PR[GP1:91,1] = PR[GP1:90,1] + 42.235;
   1:  PR[GP1:91,2] = PR[GP1:90,2] + -33.877;
   1:L PR[91] 10mm/sec CNT100;
   1:  PR[GP1:91,1] = PR[GP1:90,1] + 47.917;
   1:  PR[GP1:91,2] = PR[GP1:90,2] + -33.127;
   1:L PR[91] 10mm/sec CNT100;
   1:  PR[GP1:91,1] = PR[GP1:90,1] + 51.138;
   1:  PR[GP1:91,2] = PR[GP1:90,2] + -31.530;
   1:L PR[91] 10mm/sec CNT100;
   1:  PR[GP1:91,1] = PR[GP1:90,1] + 56.641;
   1:  PR[GP1:91,2] = PR[GP1:90,2] + -29.504;
   1:L PR[91] 10mm/sec CNT100;
   1:  PR[GP1:91,1] = PR[GP1:90,1] + 61.453;
   1:  PR[GP1:91,2] = PR[GP1:90,2] + -26.391;
   1:L PR[91] 10mm/sec CNT100;
   1:  PR[GP1:91,1] = PR[GP1:90,1] + 63.675;
   1:  PR[GP1:91,2] = PR[GP1:90,2] + -23.565;
